  MoveL 3278 to (17.58, -71, -2.56) mm, rotated rx 180 ry 0 rz 90 deg; joints [71.731, -16.979, 81.744, 0, 25.235, 71.731]
  MoveL 3279 to (18.11, -72.42, -2.97) mm, rotated rx -180 ry 0 rz 90 deg; joints [71.692, -16.939, 81.658, 0, 25.28, 71.692]
  MoveL 3280 to (18.93, -73.7, -3.38) mm, rotated rx -180 ry 0 rz 90 deg; joints [71.66, -16.893, 81.554, 0, 25.339, 71.66]
  MoveL 3281 to (20.03, -74.75, -3.78) mm, rotated rx 180 ry 0 rz 90 deg; joints [71.639, -16.843, 81.436, 0, 25.408, 71.639]
  MoveL 3282 to (21.32, -75.54, -4.19) mm, rotated rx 180 ry 0 rz 90 deg; joints [71.627, -16.791, 81.309, 0, 25.482, 71.627]
  MoveL 3283 to (22.76, -76.03, -4.59) mm, rotated rx 180 ry 0 rz 90 deg; joints [71.627, -16.738, 81.179, 0, 25.559, 71.627]
  MoveL 3284 to (24.27, -76.15, -5) mm, rotated rx -180 ry 0 rz 90 deg; joints [71.639, -16.686, 81.052, 0, 25.634, 71.639]
  MoveL 3285 to (45.96, -75.93, -5) mm, rotated rx 180 ry 0 rz 90 deg; joints [71.867, -16.234, 79.464, 0, 26.77, 71.867]
  MoveL 3286 to (52.59, -75.84, -5) mm, rotated rx -180 ry 0 rz 90 deg; joints [71.937, -16.091, 78.973, 0, 27.118, 71.937]
  MoveC 3287 to (55.58, -72.68, -5) mm, rotated rx -180 ry 0 rz 90 deg; joints [72.063, -16.048, 78.827, 0, 27.222, 72.063] to (55.72, -68.34, -5) mm, rotated rx -180 ry 0 rz 90 deg; joints [72.198, -16.076, 78.921, 0, 27.155, 72.198]
  MoveL 3288 to (51.98, -63.97, -5) mm, rotated rx 180 ry 0 rz 90 deg; joints [72.296, -16.187, 79.304, 0, 26.883, 72.296]
  MoveL 3289 to (27.4, -35.54, -5) mm, rotated rx 180 ry 0 rz 90 deg; joints [72.942, -16.885, 81.769, 0, 25.117, 72.942]
  MoveL 3290 to (27.01, -35.1, -5) mm, rotated rx 180 ry 0 rz 90 deg; joints [72.952, -16.896, 81.807, 0, 25.089, 72.952]
  MoveL 3291 to (26.45, -34.59, -5) mm, rotated rx -180 ry 0 rz 90 deg; joints [72.963, -16.91, 81.859, 0, 25.052, 72.963]
  MoveL 3292 to (20.53, -29.85, -5) mm, rotated rx 180 ry 0 rz 90 deg; joints [73.055, -17.057, 82.393, 0, 24.664, 73.055]
  MoveL 3293 to (12.79, -23.65, -5) mm, rotated rx -180 ry 0 rz 90 deg; joints [73.178, -17.244, 83.085, 0, 24.159, 73.178]
  MoveL 3294 to (11.85, -22.94, -5) mm, rotated rx -180 ry 0 rz 90 deg; joints [73.191, -17.267, 83.168, 0, 24.098, 73.191]
  MoveC 3295 to (8.28, -22.05, -5) mm, rotated rx 180 ry 0 rz 90 deg; joints [73.185, -17.34, 83.443, 0, 23.897, 73.185] to (5.13, -23.95, -5) mm, rotated rx 180 ry 0 rz 90 deg; joints [73.094, -17.389, 83.626, 0, 23.763, 73.094]
  MoveC 3296 to (4.8, -24.62, -5) mm, rotated rx -180 ry 0 rz 90 deg; joints [73.069, -17.391, 83.635, 0, 23.756, 73.069] to (4.56, -25.32, -5) mm, rotated rx 180 ry 0 rz 90 deg; joints [73.045, -17.392, 83.637, 0, 23.755, 73.045]
  MoveL 3297 to (-7.48, -70.6, -5) mm, rotated rx 180 ry 0 rz 90 deg; joints [71.481, -17.345, 83.463, 0, 23.882, 71.481]
  MoveC 3298 to (-7, -74.19, -5) mm, rotated rx -180 ry 0 rz 90 deg; joints [71.372, -17.314, 83.344, 0, 23.969, 71.372] to (-4.04, -76.29, -5) mm, rotated rx -180 ry 0 rz 90 deg; joints [71.338, -17.244, 83.084, 0, 24.16, 71.338]
  MoveC 3299 to (-3.21, -76.4, -5) mm, rotated rx 180 ry 0 rz 90 deg; joints [71.343, -17.227, 83.022, 0, 24.205, 71.343] to (-2.37, -76.42, -5) mm, rotated rx 180 ry 0 rz 90 deg; joints [71.351, -17.211, 82.962, 0, 24.249, 71.351]
  MoveL 3300 to (24.27, -76.15, -5) mm, rotated rx -180 ry 0 rz 90 deg; joints [71.639, -16.686, 81.052, 0, 25.634, 71.639]
  MoveL 3301 to (24.2, -68.6, -5) mm, rotated rx -180 ry 0 rz 90 deg; joints [71.873, -16.738, 81.239, 0, 25.5, 71.873]
  MoveL 3302 to (24.2, -68.6, -2) mm, rotated rx 180 ry 0 rz 90 deg; joints [71.873, -16.89, 81.34, 0, 25.55, 71.873]
  Establecer velocidad (1000.0 mm/s)
  MoveL 3303 to (24.2, -68.6, 10) mm, rotated rx -180 ry 0 rz 90 deg; joints [71.873, -17.496, 81.742, 0, 25.754, 71.873]
  Establecer velocidad (66.7 mm/s)
  MoveL 3304 to (66.41, -31.14, 10) mm, rotated rx 180 ry 0 rz 90 deg; joints [73.447, -16.845, 79.487, 0, 27.358, 73.447]
  MoveL 3305 to (66.41, -31.14, -1.75) mm, rotated rx -180 ry 0 rz 90 deg; joints [73.447, -16.257, 79.092, 0, 27.164, 73.447]
  MoveL 3306 to (67.91, -31.32, -2.16) mm, rotated rx -180 ry 0 rz 90 deg; joints [73.456, -16.202, 78.961, 0, 27.241, 73.456]
  MoveL 3307 to (69.42, -31.14, -2.56) mm, rotated rx 180 ry 0 rz 90 deg; joints [73.475, -16.149, 78.838, 0, 27.312, 73.475]
  MoveL 3308 to (70.85, -30.62, -2.97) mm, rotated rx 180 ry 0 rz 90 deg; joints [73.504, -16.101, 78.727, 0, 27.373, 73.504]
  MoveL 3309 to (72.13, -29.81, -3.38) mm, rotated rx -180 ry 0 rz 90 deg; joints [73.541, -16.057, 78.635, 0, 27.422, 73.541]
  MoveL 3310 to (73.2, -28.73, -3.78) mm, rotated rx 180 ry 0 rz 90 deg; joints [73.584, -16.02, 78.564, 0, 27.456, 73.584]
  MoveL 3311 to (74.01, -27.44, -4.19) mm, rotated rx -180 ry 0 rz 90 deg; joints [73.631, -15.99, 78.518, 0, 27.472, 73.631]
  MoveL 3312 to (74.51, -26, -4.59) mm, rotated rx 180 ry 0 rz 90 deg; joints [73.68, -15.968, 78.498, 0, 27.47, 73.68]
  MoveL 3313 to (74.65, -24.49, -5) mm, rotated rx -180 ry 0 rz 90 deg; joints [73.728, -15.954, 78.507, 0, 27.447, 73.728]
  MoveL 3314 to (74.64, -7.37, -5) mm, rotated rx -180 ry 0 rz 90 deg; joints [74.258, -16.064, 78.879, 0, 27.184, 74.258]
  MoveC 3315 to (72.62, -4.69, -5) mm, rotated rx 180 ry 0 rz 90 deg; joints [74.324, -16.125, 79.089, 0, 27.036, 74.324] to (69.65, -3.13, -5) mm, rotated rx -180 ry 0 rz 90 deg; joints [74.346, -16.199, 79.346, 0, 26.854, 74.346]
  MoveC 3316 to (68.13, -3, -5) mm, rotated rx 180 ry 0 rz 90 deg; joints [74.337, -16.233, 79.463, 0, 26.77, 74.337] to (66.64, -3.36, -5) mm, rotated rx -180 ry 0 rz 90 deg; joints [74.313, -16.263, 79.567, 0, 26.696, 74.313]
  MoveL 3317 to (51.96, -23.48, -5) mm, rotated rx -180 ry 0 rz 90 deg; joints [73.552, -16.454, 80.231, 0, 26.223, 73.552]
  MoveC 3318 to (51.14, -26.2, -5) mm, rotated rx -180 ry 0 rz 90 deg; joints [73.46, -16.454, 80.232, 0, 26.222, 73.46] to (52.21, -28.84, -5) mm, rotated rx 180 ry 0 rz 90 deg; joints [73.387, -16.415, 80.094, 0, 26.321, 73.387]
  MoveL 3319 to (67.07, -45.61, -5) mm, rotated rx 180 ry 0 rz 90 deg; joints [73.007, -15.983, 78.603, 0, 27.38, 73.007]
  MoveC 3320 to (69.47, -45.88, -5) mm, rotated rx 180 ry 0 rz 90 deg; joints [73.021, -15.928, 78.416, 0, 27.512, 73.021] to (71.71, -45.01, -5) mm, rotated rx 180 ry 0 rz 90 deg; joints [73.069, -15.883, 78.266, 0, 27.617, 73.069]
  MoveL 3321 to (72.16, -44.7, -5) mm, rotated rx 180 ry 0 rz 90 deg; joints [73.082, -15.875, 78.239, 0, 27.636, 73.082]
  MoveC 3322 to (73.61, -43.33, -5) mm, rotated rx 180 ry 0 rz 90 deg; joints [73.138, -15.852, 78.161, 0, 27.692, 73.138] to (74.63, -41.62, -5) mm, rotated rx 180 ry 0 rz 90 deg; joints [73.2, -15.841, 78.123, 0, 27.718, 73.2]
  MoveL 3323 to (74.65, -41.22, -5) mm, rotated rx -180 ry 0 rz 90 deg; joints [73.212, -15.843, 78.131, 0, 27.713, 73.212]
  MoveL 3324 to (74.65, -24.49, -5) mm, rotated rx -180 ry 0 rz 90 deg; joints [73.728, -15.954, 78.507, 0, 27.447, 73.728]
  MoveL 3325 to (67.09, -24.5, -5) mm, rotated rx 180 ry 0 rz 90 deg; joints [73.659, -16.121, 79.077, 0, 27.044, 73.659]
  MoveL 3326 to (67.09, -24.5, -2) mm, rotated rx -180 ry 0 rz 90 deg; joints [73.659, -16.272, 79.18, 0, 27.092, 73.659]
  Establecer velocidad (1000.0 mm/s)
  MoveL 3327 to (67.09, -24.5, 10) mm, rotated rx -180 ry 0 rz 90 deg; joints [73.659, -16.873, 79.583, 0, 27.29, 73.659]
  Establecer velocidad (66.7 mm/s)
  MoveL 3328 to (37.4, 23.7, 10) mm, rotated rx 180 ry 0 rz 90 deg; joints [74.913, -17.787, 82.786, 0, 25.001, 74.913]
  MoveL 3329 to (37.4, 23.7, -1.75) mm, rotated rx -180 ry 0 rz 90 deg; joints [74.913, -17.192, 82.393, 0, 24.798, 74.913]
  MoveL 3330 to (37.54, 25.21, -2.16) mm, rotated rx -180 ry 0 rz 90 deg; joints [74.963, -17.177, 82.399, 0, 24.778, 74.963]
  MoveL 3331 to (37.32, 26.71, -2.56) mm, rotated rx 180 ry 0 rz 90 deg; joints [75.009, -17.168, 82.431, 0, 24.738, 75.009]
  MoveL 3332 to (36.77, 28.13, -2.97) mm, rotated rx 180 ry 0 rz 90 deg; joints [75.049, -17.166, 82.485, 0, 24.682, 75.049]
  MoveL 3333 to (35.92, 29.39, -3.38) mm, rotated rx -180 ry 0 rz 90 deg; joints [75.082, -17.169, 82.557, 0, 24.612, 75.082]
  MoveL 3334 to (34.81, 30.43, -3.78) mm, rotated rx 180 ry 0 rz 90 deg; joints [75.106, -17.176, 82.645, 0, 24.531, 75.106]
  MoveL 3335 to (33.5, 31.2, -4.19) mm, rotated rx -180 ry 0 rz 90 deg; joints [75.12, -17.185, 82.741, 0, 24.444, 75.12]
  MoveL 3336 to (32.05, 31.66, -4.59) mm, rotated rx 180 ry 0 rz 90 deg; joints [75.122, -17.196, 82.841, 0, 24.354, 75.122]
  MoveL 3337 to (30.54, 31.76, -5) mm, rotated rx 180 ry 0 rz 90 deg; joints [75.113, -17.205, 82.94, 0, 24.266, 75.113]
  MoveL 3338 to (8.05, 31.16, -5) mm, rotated rx 180 ry 0 rz 90 deg; joints [74.898, -17.63, 84.544, 0, 23.085, 74.898]
  MoveL 3339 to (7.58, 31.11, -5) mm, rotated rx 180 ry 0 rz 90 deg; joints [74.893, -17.638, 84.577, 0, 23.061, 74.893]
  MoveC 3340 to (4.29, 29.28, -5) mm, rotated rx 180 ry 0 rz 90 deg; joints [74.804, -17.69, 84.776, 0, 22.914, 74.804] to (3.5, 25.59, -5) mm, rotated rx 180 ry 0 rz 90 deg; joints [74.677, -17.685, 84.76, 0, 22.925, 74.677]
  MoveL 3341 to (3.65, 25.11, -5) mm, rotated rx -180 ry 0 rz 90 deg; joints [74.663, -17.68, 84.741, 0, 22.94, 74.663]
  MoveL 3342 to (9.48, 9, -5) mm, rotated rx 180 ry 0 rz 90 deg; joints [74.194, -17.489, 84.006, 0, 23.483, 74.194]
  MoveL 3343 to (9.79, 8.22, -5) mm, rotated rx 180 ry 0 rz 90 deg; joints [74.171, -17.479, 83.968, 0, 23.511, 74.171]
  MoveC 3344 to (10.34, 7.22, -5) mm, rotated rx -180 ry 0 rz 90 deg; joints [74.144, -17.463, 83.908, 0, 23.555, 74.144] to (11.15, 6.4, -5) mm, rotated rx 180 ry 0 rz 90 deg; joints [74.125, -17.444, 83.834, 0, 23.61, 74.125]
  MoveL 3345 to (27.96, -6.68, -5) mm, rotated rx 180 ry 0 rz 90 deg; joints [73.861, -17.046, 82.353, 0, 24.693, 73.861]
  MoveL 3346 to (28.63, -7.18, -5) mm, rotated rx -180 ry 0 rz 90 deg; joints [73.851, -17.03, 82.294, 0, 24.736, 73.851]
  MoveC 3347 to (31.82, -7.71, -5) mm, rotated rx 180 ry 0 rz 90 deg; joints [73.864, -16.963, 82.05, 0, 24.913, 73.864] to (34.59, -6.03, -5) mm, rotated rx 180 ry 0 rz 90 deg; joints [73.942, -16.917, 81.884, 0, 25.034, 73.942]
  MoveL 3348 to (35.19, -5.21, -5) mm, rotated rx -180 ry 0 rz 90 deg; joints [73.974, -16.91, 81.857, 0, 25.053, 73.974]
  MoveL 3349 to (55.44, 23.03, -5) mm, rotated rx 180 ry 0 rz 90 deg; joints [75.046, -16.655, 80.943, 0, 25.713, 75.046]
  MoveL 3350 to (56.93, 25.11, -5) mm, rotated rx 180 ry 0 rz 90 deg; joints [75.124, -16.636, 80.873, 0, 25.762, 75.124]
  MoveC 3351 to (56.59, 29.37, -5) mm, rotated rx 180 ry 0 rz 90 deg; joints [75.256, -16.666, 80.982, 0, 25.684, 75.256] to (53.5, 32.33, -5) mm, rotated rx -180 ry 0 rz 90 deg; joints [75.325, -16.747, 81.268, 0, 25.478, 75.325]
  MoveL 3352 to (49.75, 32.27, -5) mm, rotated rx -180 ry 0 rz 90 deg; joints [75.291, -16.823, 81.544, 0, 25.279, 75.291]
  MoveL 3353 to (30.54, 31.76, -5) mm, rotated rx 180 ry 0 rz 90 deg; joints [75.113, -17.205, 82.94, 0, 24.266, 75.113]
  MoveL 3354 to (30.74, 24.21, -5) mm, rotated rx -180 ry 0 rz 90 deg; joints [74.872, -17.162, 82.778, 0, 24.383, 74.872]
  MoveL 3355 to (30.74, 24.21, -2) mm, rotated rx -180 ry 0 rz 90 deg; joints [74.872, -17.314, 82.88, 0, 24.434, 74.872]
  Establecer velocidad (1000.0 mm/s)
  MoveL 3356 to (30.74, 24.21, 10) mm, rotated rx -180 ry 0 rz 90 deg; joints [74.872, -17.923, 83.28, 0, 24.643, 74.872]
  Establecer velocidad (66.7 mm/s)
  MoveL 3357 to (25.69, 67.74, 10) mm, rotated rx 180 ry 0 rz 90 deg; joints [76.236, -18.241, 84.456, 0, 23.784, 76.236]
  MoveL 3358 to (25.69, 67.74, -1.75) mm, rotated rx -180 ry 0 rz 90 deg; joints [76.236, -17.642, 84.065, 0, 23.577, 76.236]
  MoveL 3359 to (25.89, 69.24, -2.16) mm, rotated rx -180 ry 0 rz 90 deg; joints [76.287, -17.624, 84.063, 0, 23.561, 76.287]
  MoveL 3360 to (25.73, 70.75, -2.56) mm, rotated rx 180 ry 0 rz 90 deg; joints [76.335, -17.613, 84.088, 0, 23.525, 76.335]
  MoveL 3361 to (25.23, 72.19, -2.97) mm, rotated rx -180 ry 0 rz 90 deg; joints [76.378, -17.609, 84.135, 0, 23.474, 76.378]
  MoveL 3362 to (24.43, 73.48, -3.38) mm, rotated rx 180 ry 0 rz 90 deg; joints [76.413, -17.609, 84.202, 0, 23.407, 76.413]
  MoveL 3363 to (23.36, 74.56, -3.78) mm, rotated rx -180 ry 0 rz 90 deg; joints [76.44, -17.613, 84.284, 0, 23.33, 76.44]
  MoveL 3364 to (22.08, 75.38, -4.19) mm, rotated rx 180 ry 0 rz 90 deg; joints [76.457, -17.62, 84.376, 0, 23.244, 76.457]
  MoveL 3365 to (20.65, 75.89, -4.59) mm, rotated rx -180 ry 0 rz 90 deg; joints [76.463, -17.629, 84.474, 0, 23.155, 76.463]
  MoveL 3366 to (19.14, 76.05, -5) mm, rotated rx -180 ry 0 rz 90 deg; joints [76.456, -17.637, 84.571, 0, 23.065, 76.456]
  MoveL 3367 to (-29.85, 76.54, -5) mm, rotated rx 180 ry 0 rz 90 deg; joints [76.075, -18.492, 88.024, 0, 20.469, 76.075]
  MoveL 3368 to (-31.98, 76.46, -5) mm, rotated rx 180 ry 0 rz 90 deg; joints [76.054, -18.527, 88.169, 0, 20.357, 76.054]
  MoveC 3369 to (-34.9, 72.87, -5) mm, rotated rx 180 ry 0 rz 90 deg; joints [75.909, -18.559, 88.309, 0, 20.251, 75.909] to (-34.36, 68.26, -5) mm, rotated rx 180 ry 0 rz 90 deg; joints [75.758, -18.532, 88.191, 0, 20.341, 75.758]
  MoveL 3370 to (-33.58, 67.76, -5) mm, rotated rx -180 ry 0 rz 90 deg; joints [75.748, -18.517, 88.129, 0, 20.388, 75.748]
  MoveL 3371 to (-11.56, 53.8, -5) mm, rotated rx 180 ry 0 rz 90 deg; joints [75.471, -18.088, 86.352, 0, 21.736, 75.471]
  MoveC 3372 to (-9.41, 52.87, -5) mm, rotated rx 180 ry 0 rz 90 deg; joints [75.459, -18.047, 86.185, 0, 21.862, 75.459] to (-7.08, 52.65, -5) mm, rotated rx 180 ry 0 rz 90 deg; joints [75.471, -18.005, 86.017, 0, 21.988, 75.471]
  MoveL 3373 to (-6.16, 52.71, -5) mm, rotated rx 180 ry 0 rz 90 deg; joints [75.481, -17.989, 85.953, 0, 22.035, 75.481]
  MoveL 3374 to (56.39, 57.32, -5) mm, rotated rx -180 ry 0 rz 90 deg; joints [76.144, -16.818, 81.525, 0, 25.293, 76.144]
  MoveL 3375 to (69.65, 58.51, -5) mm, rotated rx -180 ry 0 rz 90 deg; joints [76.285, -16.547, 80.559, 0, 25.988, 76.285]
  MoveL 3376 to (70.5, 58.62, -5) mm, rotated rx -180 ry 0 rz 90 deg; joints [76.295, -16.53, 80.497, 0, 26.032, 76.295]
  MoveC 3377 to (72.99, 59.89, -5) mm, rotated rx 180 ry 0 rz 90 deg; joints [76.355, -16.483, 80.334, 0, 26.149, 76.355] to (74.04, 62.48, -5) mm, rotated rx 180 ry 0 rz 90 deg; joints [76.445, -16.474, 80.302, 0, 26.172, 76.445]
  MoveL 3378 to (74.05, 63.02, -5) mm, rotated rx -180 ry 0 rz 90 deg; joints [76.462, -16.477, 80.311, 0, 26.166, 76.462]
  MoveL 3379 to (74.05, 70.6, -5) mm, rotated rx 180 ry 0 rz 90 deg; joints [76.703, -16.515, 80.447, 0, 26.068, 76.703]
  MoveL 3380 to (74.03, 71.11, -5) mm, rotated rx 180 ry 0 rz 90 deg; joints [76.719, -16.518, 80.457, 0, 26.061, 76.719]
  MoveC 3381 to (72.87, 73.73, -5) mm, rotated rx -180 ry 0 rz 90 deg; joints [76.793, -16.556, 80.591, 0, 25.965, 76.793] to (70.25, 74.88, -5) mm, rotated rx -180 ry 0 rz 90 deg; joints [76.81, -16.617, 80.808, 0, 25.81, 76.81]
  MoveC 3382 to (46.61, 75.6, -5) mm, rotated rx 180 ry 0 rz 90 deg; joints [76.655, -17.106, 82.572, 0, 24.534, 76.655] to (22.97, 76, -5) mm, rotated rx -180 ry 0 rz 90 deg; joints [76.485, -17.565, 84.296, 0, 23.269, 76.485]
  MoveL 3383 to (19.14, 76.05, -5) mm, rotated rx -180 ry 0 rz 90 deg; joints [76.456, -17.637, 84.571, 0, 23.065, 76.456]
  MoveL 3384 to (19.06, 68.5, -5) mm, rotated rx -180 ry 0 rz 90 deg; joints [76.208, -17.604, 84.445, 0, 23.159, 76.208]
  MoveL 3385 to (19.06, 68.5, -2) mm, rotated rx -180 ry 0 rz 90 deg; joints [76.208, -17.757, 84.547, 0, 23.211, 76.208]
  Establecer velocidad (1000.0 mm/s)
  MoveL 3386 to (19.06, 68.5, 10) mm, rotated rx -180 ry 0 rz 90 deg; joints [76.208, -18.37, 84.946, 0, 23.424, 76.208]
  Establecer velocidad (66.7 mm/s)
  MoveL 3387 to (25.69, 67.49, 10) mm, rotated rx -180 ry 0 rz 90 deg; joints [76.228, -18.239, 84.452, 0, 23.788, 76.228]
  MoveL 3388 to (25.69, 67.49, -2) mm, rotated rx -180 ry 0 rz 90 deg; joints [76.228, -17.628, 84.052, 0, 23.576, 76.228]
  MoveL 3389 to (25.89, 68.99, -2.41) mm, rotated rx 180 ry 0 rz 90 deg; joints [76.279, -17.61, 84.05, 0, 23.56, 76.279]
  MoveL 3390 to (25.73, 70.51, -2.81) mm, rotated rx -180 ry 0 rz 90 deg; joints [76.327, -17.6, 84.075, 0, 23.524, 76.327]
  MoveL 3391 to (25.23, 71.94, -3.22) mm, rotated rx -180 ry 0 rz 90 deg; joints [76.37, -17.595, 84.123, 0, 23.472, 76.37]
  MoveL 3392 to (24.42, 73.23, -3.62) mm, rotated rx -180 ry 0 rz 90 deg; joints [76.405, -17.595, 84.189, 0, 23.406, 76.405]
  MoveL 3393 to (23.36, 74.31, -4.03) mm, rotated rx 180 ry 0 rz 90 deg; joints [76.432, -17.6, 84.271, 0, 23.328, 76.432]
  MoveL 3394 to (22.08, 75.13, -4.44) mm, rotated rx 180 ry 0 rz 90 deg; joints [76.449, -17.606, 84.364, 0, 23.243, 76.449]
  MoveL 3395 to (20.65, 75.64, -4.84) mm, rotated rx 180 ry 0 rz 90 deg; joints [76.454, -17.615, 84.462, 0, 23.153, 76.454]
  MoveL 3396 to (19.14, 75.8, -5.25) mm, rotated rx 180 ry 0 rz 90 deg; joints [76.448, -17.623, 84.559, 0, 23.064, 76.448]
  MoveL 3397 to (-25.11, 76.24, -5.25) mm, rotated rx -180 ry 0 rz 90 deg; joints [76.104, -18.401, 87.683, 0, 20.718, 76.104]
  MoveL 3398 to (-30.8, 76.27, -5.25) mm, rotated rx 180 ry 0 rz 90 deg; joints [76.058, -18.494, 88.076, 0, 20.418, 76.058]
  MoveL 3399 to (-31.4, 76.24, -5.25) mm, rotated rx 180 ry 0 rz 90 deg; joints [76.052, -18.504, 88.117, 0, 20.386, 76.052]
  MoveC 3400 to (-34.26, 72.7, -5.25) mm, rotated rx 180 ry 0 rz 90 deg; joints [75.908, -18.535, 88.253, 0, 20.282, 75.908] to (-33.75, 68.18, -5.25) mm, rotated rx 180 ry 0 rz 90 deg; joints [75.761, -18.509, 88.14, 0, 20.369, 75.761]
  MoveL 3401 to (-33.1, 67.76, -5.25) mm, rotated rx -180 ry 0 rz 90 deg; joints [75.752, -18.497, 88.088, 0, 20.409, 75.752]
  MoveL 3402 to (-11.42, 54, -5.25) mm, rotated rx -180 ry 0 rz 90 deg; joints [75.479, -18.074, 86.337, 0, 21.736, 75.479]
  MoveC 3403 to (-9.3, 53.09, -5.25) mm, rotated rx 180 ry 0 rz 90 deg; joints [75.467, -18.033, 86.172, 0, 21.86, 75.467] to (-7, 52.9, -5.25) mm, rotated rx -180 ry 0 rz 90 deg; joints [75.48, -17.992, 86.007, 0, 21.984, 75.48]
  MoveL 3404 to (45.99, 56.79, -5.25) mm, rotated rx -180 ry 0 rz 90 deg; joints [76.044, -17.014, 82.274, 0, 24.74, 76.044]
  MoveC 3405 to (57.83, 57.75, -5.25) mm, rotated rx 180 ry 0 rz 90 deg; joints [76.169, -16.778, 81.418, 0, 25.36, 76.169] to (69.65, 58.87, -5.25) mm, rotated rx 180 ry 0 rz 90 deg; joints [76.297, -16.536, 80.557, 0, 25.979, 76.297]
  MoveL 3406 to (70.41, 58.98, -5.25) mm, rotated rx 180 ry 0 rz 90 deg; joints [76.306, -16.521, 80.503, 0, 26.018, 76.306]
  MoveC 3407 to (72.7, 60.18, -5.25) mm, rotated rx 180 ry 0 rz 90 deg; joints [76.362, -16.478, 80.352, 0, 26.126, 76.362] to (73.71, 62.58, -5.25) mm, rotated rx -180 ry 0 rz 90 deg; joints [76.445, -16.469, 80.32, 0, 26.149, 76.445]
  MoveL 3408 to (73.73, 63.02, -5.25) mm, rotated rx -180 ry 0 rz 90 deg; joints [76.46, -16.471, 80.326, 0, 26.145, 76.46]
  MoveL 3409 to (73.73, 70.6, -5.25) mm, rotated rx -180 ry 0 rz 90 deg; joints [76.7, -16.509, 80.462, 0, 26.047, 76.7]
  MoveL 3410 to (73.7, 71.06, -5.25) mm, rotated rx 180 ry 0 rz 90 deg; joints [76.715, -16.513, 80.473, 0, 26.039, 76.715]
  MoveC 3411 to (72.55, 73.49, -5.25) mm, rotated rx 180 ry 0 rz 90 deg; joints [76.783, -16.549, 80.602, 0, 25.947, 76.783] to (70.08, 74.55, -5.25) mm, rotated rx 180 ry 0 rz 90 deg; joints [76.799, -16.607, 80.806, 0, 25.801, 76.799]
  MoveC 3412 to (44.76, 75.38, -5.25) mm, rotated rx 180 ry 0 rz 90 deg; joints [76.633, -17.129, 82.695, 0, 24.434, 76.633] to (19.43, 75.79, -5.25) mm, rotated rx -180 ry 0 rz 90 deg; joints [76.45, -17.617, 84.538, 0, 23.08, 76.45]
  MoveL 3413 to (19.14, 75.8, -5.25) mm, rotated rx 180 ry 0 rz 90 deg; joints [76.448, -17.623, 84.559, 0, 23.064, 76.448]
  MoveL 3414 to (19.06, 68.25, -5.25) mm, rotated rx 180 ry 0 rz 90 deg; joints [76.2, -17.59, 84.432, 0, 23.158, 76.2]
  MoveL 3415 to (19.06, 68.25, -2.25) mm, rotated rx -180 ry 0 rz 90 deg; joints [76.2, -17.743, 84.534, 0, 23.21, 76.2]
  Establecer velocidad (1000.0 mm/s)
  MoveL 3416 to (19.06, 68.25, 10) mm, rotated rx -180 ry 0 rz 90 deg; joints [76.2, -18.369, 84.942, 0, 23.427, 76.2]
  Establecer velocidad (66.7 mm/s)
  MoveL 3417 to (37.41, 23.42, 10) mm, rotated rx 180 ry 0 rz 90 deg; joints [74.905, -17.785, 82.78, 0, 25.006, 74.905]
  MoveL 3418 to (37.41, 23.42, -2) mm, rotated rx 180 ry 0 rz 90 deg; joints [74.905, -17.178, 82.379, 0, 24.799, 74.905]
  MoveL 3419 to (37.56, 24.93, -2.41) mm, rotated rx 180 ry 0 rz 90 deg; joints [74.954, -17.162, 82.384, 0, 24.778, 74.954]
  MoveL 3420 to (37.33, 26.44, -2.81) mm, rotated rx 180 ry 0 rz 90 deg; joints [75, -17.154, 82.416, 0, 24.738, 75]
  MoveL 3421 to (36.78, 27.85, -3.22) mm, rotated rx 180 ry 0 rz 90 deg; joints [75.041, -17.152, 82.47, 0, 24.682, 75.041]
  MoveL 3422 to (35.94, 29.11, -3.62) mm, rotated rx -180 ry 0 rz 90 deg; joints [75.074, -17.155, 82.543, 0, 24.612, 75.074]
  MoveL 3423 to (34.83, 30.15, -4.03) mm, rotated rx 180 ry 0 rz 90 deg; joints [75.098, -17.162, 82.63, 0, 24.532, 75.098]
  MoveL 3424 to (33.52, 30.92, -4.44) mm, rotated rx 180 ry 0 rz 90 deg; joints [75.111, -17.171, 82.726, 0, 24.445, 75.111]
  MoveL 3425 to (32.07, 31.39, -4.84) mm, rotated rx 180 ry 0 rz 90 deg; joints [75.114, -17.181, 82.827, 0, 24.354, 75.114]
  MoveL 3426 to (30.56, 31.49, -5.25) mm, rotated rx 180 ry 0 rz 90 deg; joints [75.104, -17.191, 82.925, 0, 24.266, 75.104]
  MoveL 3427 to (8.05, 30.9, -5.25) mm, rotated rx 180 ry 0 rz 90 deg; joints [74.89, -17.616, 84.531, 0, 23.085, 74.89]
  MoveC 3428 to (4.7, 29.22, -5.25) mm, rotated rx 180 ry 0 rz 90 deg; joints [74.806, -17.669, 84.737, 0, 22.932, 74.806] to (3.77, 25.59, -5.25) mm, rotated rx -180 ry 0 rz 90 deg; joints [74.679, -17.668, 84.733, 0, 22.935, 74.679]
  MoveL 3429 to (3.92, 25.11, -5.25) mm, rotated rx 180 ry 0 rz 90 deg; joints [74.665, -17.663, 84.713, 0, 22.95, 74.665]
  MoveL 3430 to (9.96, 8.47, -5.25) mm, rotated rx 180 ry 0 rz 90 deg; joints [74.181, -17.464, 83.952, 0, 23.512, 74.181]
  MoveC 3431 to (10.51, 7.43, -5.25) mm, rotated rx 180 ry 0 rz 90 deg; joints [74.152, -17.448, 83.892, 0, 23.557, 74.152] to (11.34, 6.58, -5.25) mm, rotated rx 180 ry 0 rz 90 deg; joints [74.132, -17.428, 83.816, 0, 23.613, 74.132]
  MoveL 3432 to (27.71, -6.16, -5.25) mm, rotated rx 180 ry 0 rz 90 deg; joints [73.875, -17.041, 82.373, 0, 24.668, 73.875]
  MoveL 3433 to (27.96, -6.35, -5.25) mm, rotated rx -180 ry 0 rz 90 deg; joints [73.871, -17.035, 82.351, 0, 24.684, 73.871]
  MoveL 3434 to (28.9, -7.03, -5.25) mm, rotated rx -180 ry 0 rz 90 deg; joints [73.858, -17.013, 82.268, 0, 24.744, 73.858]
  MoveC 3435 to (32, -7.33, -5.25) mm, rotated rx -180 ry 0 rz 90 deg; joints [73.877, -16.949, 82.037, 0, 24.912, 73.877] to (34.59, -5.61, -5.25) mm, rotated rx 180 ry 0 rz 90 deg; joints [73.956, -16.907, 81.884, 0, 25.023, 73.956]
  MoveL 3436 to (55.44, 23.47, -5.25) mm, rotated rx 180 ry 0 rz 90 deg; joints [75.06, -16.645, 80.943, 0, 25.702, 75.06]
  MoveL 3437 to (56.39, 24.8, -5.25) mm, rotated rx 180 ry 0 rz 90 deg; joints [75.11, -16.633, 80.899, 0, 25.734, 75.11]
  MoveC 3438 to (56.71, 26.56, -5.25) mm, rotated rx 180 ry 0 rz 90 deg; joints [75.168, -16.636, 80.91, 0, 25.726, 75.168] to (56.39, 28.32, -5.25) mm, rotated rx -180 ry 0 rz 90 deg; joints [75.221, -16.652, 80.968, 0, 25.684, 75.221]
  MoveC 3439 to (55.15, 30.57, -5.25) mm, rotated rx -180 ry 0 rz 90 deg; joints [75.282, -16.69, 81.103, 0, 25.587, 75.282] to (53.06, 32.06, -5.25) mm, rotated rx 180 ry 0 rz 90 deg; joints [75.312, -16.742, 81.287, 0, 25.454, 75.312]
  MoveL 3440 to (52.59, 32.06, -5.25) mm, rotated rx 180 ry 0 rz 90 deg; joints [75.308, -16.751, 81.322, 0, 25.429, 75.308]
  MoveL 3441 to (30.56, 31.49, -5.25) mm, rotated rx 180 ry 0 rz 90 deg; joints [75.104, -17.191, 82.925, 0, 24.266, 75.104]
  MoveL 3442 to (30.75, 23.94, -5.25) mm, rotated rx 180 ry 0 rz 90 deg; joints [74.863, -17.147, 82.764, 0, 24.384, 74.863]
  MoveL 3443 to (30.75, 23.94, -2.25) mm, rotated rx 180 ry 0 rz 90 deg; joints [74.863, -17.3, 82.865, 0, 24.435, 74.863]
  Establecer velocidad (1000.0 mm/s)
  MoveL 3444 to (30.75, 23.94, 10) mm, rotated rx 180 ry 0 rz 90 deg; joints [74.863, -17.921, 83.274, 0, 24.647, 74.863]
  Establecer velocidad (66.7 mm/s)
  MoveL 3445 to (66.13, -31.19, 10) mm, rotated rx 180 ry 0 rz 90 deg; joints [73.443, -16.851, 79.507, 0, 27.344, 73.443]
  MoveL 3446 to (66.13, -31.19, -2) mm, rotated rx -180 ry 0 rz 90 deg; joints [73.443, -16.25, 79.103, 0, 27.147, 73.443]
  MoveL 3447 to (67.64, -31.38, -2.41) mm, rotated rx 180 ry 0 rz 90 deg; joints [73.451, -16.195, 78.972, 0, 27.223, 73.451]
  MoveL 3448 to (69.15, -31.2, -2.81) mm, rotated rx -180 ry 0 rz 90 deg; joints [73.471, -16.142, 78.848, 0, 27.294, 73.471]
  MoveL 3449 to (70.58, -30.68, -3.22) mm, rotated rx -180 ry 0 rz 90 deg; joints [73.5, -16.094, 78.738, 0, 27.356, 73.5]
  MoveL 3450 to (71.86, -29.87, -3.62) mm, rotated rx 180 ry 0 rz 90 deg; joints [73.537, -16.05, 78.646, 0, 27.405, 73.537]
  MoveL 3451 to (72.93, -28.79, -4.03) mm, rotated rx 180 ry 0 rz 90 deg; joints [73.58, -16.013, 78.575, 0, 27.438, 73.58]
  MoveL 3452 to (73.73, -27.5, -4.44) mm, rotated rx 180 ry 0 rz 90 deg; joints [73.627, -15.983, 78.529, 0, 27.455, 73.627]
  MoveL 3453 to (74.23, -26.06, -4.84) mm, rotated rx 180 ry 0 rz 90 deg; joints [73.676, -15.961, 78.509, 0, 27.452, 73.676]
  MoveL 3454 to (74.37, -24.55, -5.25) mm, rotated rx 180 ry 0 rz 90 deg; joints [73.723, -15.948, 78.518, 0, 27.43, 73.723]
  MoveL 3455 to (74.37, -8.1, -5.25) mm, rotated rx -180 ry 0 rz 90 deg; joints [74.233, -16.053, 78.876, 0, 27.177, 74.233]
  MoveC 3456 to (72.46, -5.5, -5.25) mm, rotated rx -180 ry 0 rz 90 deg; joints [74.297, -16.111, 79.075, 0, 27.035, 74.297] to (69.65, -3.92, -5.25) mm, rotated rx 180 ry 0 rz 90 deg; joints [74.322, -16.182, 79.321, 0, 26.861, 74.322]
  MoveC 3457 to (68.05, -3.71, -5.25) mm, rotated rx -180 ry 0 rz 90 deg; joints [74.314, -16.218, 79.446, 0, 26.773, 74.314] to (66.47, -4.06, -5.25) mm, rotated rx 180 ry 0 rz 90 deg; joints [74.29, -16.25, 79.557, 0, 26.694, 74.29]
  MoveL 3458 to (66.33, -4.24, -5.25) mm, rotated rx 180 ry 0 rz 90 deg; joints [74.283, -16.252, 79.563, 0, 26.689, 74.283]
  MoveL 3459 to (52.27, -23.5, -5.25) mm, rotated rx -180 ry 0 rz 90 deg; joints [73.555, -16.434, 80.199, 0, 26.236, 73.555]
  MoveC 3460 to (51.46, -26.19, -5.25) mm, rotated rx 180 ry 0 rz 90 deg; joints [73.463, -16.435, 80.199, 0, 26.235, 73.463] to (52.53, -28.79, -5.25) mm, rotated rx 180 ry 0 rz 90 deg; joints [73.392, -16.396, 80.063, 0, 26.333, 73.392]
  MoveL 3461 to (54.31, -30.8, -5.25) mm, rotated rx -180 ry 0 rz 90 deg; joints [73.346, -16.345, 79.886, 0, 26.459, 73.346]
  MoveL 3462 to (66.48, -44.54, -5.25) mm, rotated rx 180 ry 0 rz 90 deg; joints [73.034, -15.99, 78.664, 0, 27.327, 73.034]
  MoveL 3463 to (66.91, -45.01, -5.25) mm, rotated rx -180 ry 0 rz 90 deg; joints [73.024, -15.978, 78.62, 0, 27.357, 73.024]
  MoveC 3464 to (69.16, -45.22, -5.25) mm, rotated rx -180 ry 0 rz 90 deg; joints [73.038, -15.926, 78.445, 0, 27.481, 73.038] to (71.31, -44.49, -5.25) mm, rotated rx 180 ry 0 rz 90 deg; joints [73.081, -15.883, 78.3, 0, 27.583, 73.081]
  MoveC 3465 to (73.1, -42.99, -5.25) mm, rotated rx 180 ry 0 rz 90 deg; joints [73.144, -15.853, 78.199, 0, 27.655, 73.144] to (74.35, -41.01, -5.25) mm, rotated rx 180 ry 0 rz 90 deg; joints [73.216, -15.839, 78.149, 0, 27.689, 73.216]
  MoveL 3466 to (74.37, -40.27, -5.25) mm, rotated rx -180 ry 0 rz 90 deg; joints [73.239, -15.843, 78.165, 0, 27.679, 73.239]
  MoveL 3467 to (74.37, -24.55, -5.25) mm, rotated rx 180 ry 0 rz 90 deg; joints [73.723, -15.948, 78.518, 0, 27.43, 73.723]
  MoveL 3468 to (66.82, -24.55, -5.25) mm, rotated rx -180 ry 0 rz 90 deg; joints [73.655, -16.114, 79.088, 0, 27.026, 73.655]
  MoveL 3469 to (66.82, -24.55, -2.25) mm, rotated rx 180 ry 0 rz 90 deg; joints [73.655, -16.265, 79.19, 0, 27.075, 73.655]
  Establecer velocidad (1000.0 mm/s)
  MoveL 3470 to (66.82, -24.55, 10) mm, rotated rx 180 ry 0 rz 90 deg; joints [73.655, -16.879, 79.602, 0, 27.277, 73.655]
  Establecer velocidad (66.7 mm/s)
  MoveL 3471 to (17.59, -67.73, 10) mm, rotated rx 180 ry 0 rz 90 deg; joints [71.833, -17.636, 82.242, 0, 25.394, 71.833]
  MoveL 3472 to (17.59, -67.73, -2) mm, rotated rx -180 ry 0 rz 90 deg; joints [71.833, -17.029, 81.84, 0, 25.189, 71.833]
  MoveL 3473 to (17.42, -69.24, -2.41) mm, rotated rx -180 ry 0 rz 90 deg; joints [71.784, -17.002, 81.803, 0, 25.199, 71.784]
  MoveL 3474 to (17.61, -70.74, -2.81) mm, rotated rx -180 ry 0 rz 90 deg; joints [71.739, -16.968, 81.739, 0, 25.228, 71.739]
  MoveL 3475 to (18.14, -72.17, -3.22) mm, rotated rx -180 ry 0 rz 90 deg; joints [71.7, -16.927, 81.653, 0, 25.274, 71.7]
  MoveL 3476 to (18.97, -73.44, -3.62) mm, rotated rx 180 ry 0 rz 90 deg; joints [71.669, -16.881, 81.549, 0, 25.332, 71.669]
  MoveL 3477 to (20.06, -74.5, -4.03) mm, rotated rx -180 ry 0 rz 90 deg; joints [71.647, -16.832, 81.431, 0, 25.401, 71.647]
  MoveL 3478 to (21.36, -75.29, -4.44) mm, rotated rx -180 ry 0 rz 90 deg; joints [71.636, -16.78, 81.304, 0, 25.476, 71.636]
  MoveL 3479 to (22.8, -75.78, -4.84) mm, rotated rx 180 ry 0 rz 90 deg; joints [71.635, -16.727, 81.174, 0, 25.553, 71.635]
  MoveL 3480 to (24.31, -75.9, -5.25) mm, rotated rx -180 ry 0 rz 90 deg; joints [71.647, -16.674, 81.047, 0, 25.627, 71.647]
  MoveL 3481 to (42.17, -75.72, -5.25) mm, rotated rx 180 ry 0 rz 90 deg; joints [71.835, -16.304, 79.741, 0, 26.562, 71.835]
  MoveL 3482 to (52.12, -75.59, -5.25) mm, rotated rx 180 ry 0 rz 90 deg; joints [71.94, -16.09, 79.006, 0, 27.085, 71.94]
  MoveC 3483 to (55.04, -72.48, -5.25) mm, rotated rx -180 ry 0 rz 90 deg; joints [72.064, -16.049, 78.863, 0, 27.186, 72.064] to (55.24, -68.23, -5.25) mm, rotated rx 180 ry 0 rz 90 deg; joints [72.197, -16.074, 78.951, 0, 27.124, 72.197]
  MoveL 3484 to (54.92, -67.79, -5.25) mm, rotated rx -180 ry 0 rz 90 deg; joints [72.207, -16.084, 78.985, 0, 27.099, 72.207]
  MoveL 3485 to (53.26, -65.86, -5.25) mm, rotated rx -180 ry 0 rz 90 deg; joints [72.25, -16.134, 79.155, 0, 26.979, 72.25]
  MoveL 3486 to (50.82, -63.02, -5.25) mm, rotated rx 180 ry 0 rz 90 deg; joints [72.314, -16.206, 79.405, 0, 26.802, 72.314]
  MoveL 3487 to (27.08, -35.54, -5.25) mm, rotated rx -180 ry 0 rz 90 deg; joints [72.939, -16.879, 81.783, 0, 25.096, 72.939]
  MoveL 3488 to (27.01, -35.47, -5.25) mm, rotated rx 180 ry 0 rz 90 deg; joints [72.94, -16.881, 81.79, 0, 25.091, 72.94]
  MoveC 3489 to (26.13, -34.67, -5.25) mm, rotated rx 180 ry 0 rz 90 deg; joints [72.957, -16.904, 81.872, 0, 25.032, 72.957] to (25.21, -33.91, -5.25) mm, rotated rx -180 ry 0 rz 90 deg; joints [72.972, -16.927, 81.955, 0, 24.972, 72.972]
  MoveL 3490 to (12.79, -23.97, -5.25) mm, rotated rx 180 ry 0 rz 90 deg; joints [73.168, -17.23, 83.069, 0, 24.16, 73.168]
  MoveL 3491 to (11.85, -23.25, -5.25) mm, rotated rx 180 ry 0 rz 90 deg; joints [73.181, -17.252, 83.153, 0, 24.099, 73.181]
  MoveC 3492 to (8.1, -22.43, -5.25) mm, rotated rx 180 ry 0 rz 90 deg; joints [73.171, -17.329, 83.439, 0, 23.889, 73.171] to (5.03, -24.74, -5.25) mm, rotated rx 180 ry 0 rz 90 deg; joints [73.068, -17.373, 83.608, 0, 23.766, 73.068]
  MoveL 3493 to (4.9, -25.11, -5.25) mm, rotated rx -180 ry 0 rz 90 deg; joints [73.055, -17.374, 83.609, 0, 23.764, 73.055]
  MoveL 3494 to (3.32, -31, -5.25) mm, rotated rx 180 ry 0 rz 90 deg; joints [72.851, -17.369, 83.593, 0, 23.776, 72.851]
  MoveL 3495 to (-7.22, -70.63, -5.25) mm, rotated rx -180 ry 0 rz 90 deg; joints [71.483, -17.328, 83.436, 0, 23.892, 71.483]
  MoveC 3496 to (-6.61, -74.22, -5.25) mm, rotated rx 180 ry 0 rz 90 deg; joints [71.376, -17.293, 83.308, 0, 23.986, 71.376] to (-3.5, -76.1, -5.25) mm, rotated rx -180 ry 0 rz 90 deg; joints [71.35, -17.222, 83.042, 0, 24.18, 71.35]
  MoveL 3497 to (-2.92, -76.16, -5.25) mm, rotated rx -180 ry 0 rz 90 deg; joints [71.354, -17.211, 82.999, 0, 24.211, 71.354]
  MoveL 3498 to (-2.37, -76.17, -5.25) mm, rotated rx 180 ry 0 rz 90 deg; joints [71.359, -17.2, 82.96, 0, 24.24, 71.359]
  MoveL 3499 to (24.31, -75.9, -5.25) mm, rotated rx -180 ry 0 rz 90 deg; joints [71.647, -16.674, 81.047, 0, 25.627, 71.647]
  MoveL 3500 to (24.23, -68.35, -5.25) mm, rotated rx 180 ry 0 rz 90 deg; joints [71.882, -16.727, 81.234, 0, 25.493, 71.882]
  MoveL 3501 to (24.23, -68.35, -2.25) mm, rotated rx 180 ry 0 rz 90 deg; joints [71.882, -16.878, 81.336, 0, 25.543, 71.882]
  Establecer velocidad (1000.0 mm/s)
  MoveL 3502 to (24.23, -68.35, 10) mm, rotated rx -180 ry 0 rz 90 deg; joints [71.882, -17.497, 81.745, 0, 25.751, 71.882]
  Establecer velocidad (66.7 mm/s)
  MoveL 3503 to (-33.52, -52.29, 10) mm, rotated rx -180 ry 0 rz 90 deg; joints [71.79, -18.698, 86.211, 0, 22.487, 71.79]
  MoveL 3504 to (-33.52, -52.29, -2) mm, rotated rx 180 ry 0 rz 90 deg; joints [71.79, -18.082, 85.812, 0, 22.27, 71.79]
  MoveL 3505 to (-32.11, -52.85, -2.41) mm, rotated rx -180 ry 0 rz 90 deg; joints [71.787, -18.033, 85.688, 0, 22.346, 71.787]
  MoveL 3506 to (-30.6, -53.06, -2.81) mm, rotated rx 180 ry 0 rz 90 deg; joints [71.796, -17.985, 85.565, 0, 22.42, 71.796]
  MoveL 3507 to (-29.09, -52.92, -3.22) mm, rotated rx -180 ry 0 rz 90 deg; joints [71.817, -17.938, 85.45, 0, 22.489, 71.817]
  MoveL 3508 to (-27.64, -52.45, -3.62) mm, rotated rx 180 ry 0 rz 90 deg; joints [71.847, -17.894, 85.346, 0, 22.548, 71.847]
  MoveL 3509 to (-26.33, -51.68, -4.03) mm, rotated rx 180 ry 0 rz 90 deg; joints [71.886, -17.855, 85.259, 0, 22.596, 71.886]
  MoveL 3510 to (-25.23, -50.63, -4.44) mm, rotated rx -180 ry 0 rz 90 deg; joints [71.931, -17.82, 85.192, 0, 22.628, 71.931]
  MoveL 3511 to (-24.38, -49.37, -4.84) mm, rotated rx 180 ry 0 rz 90 deg; joints [71.981, -17.792, 85.148, 0, 22.644, 71.981]
  MoveL 3512 to (-23.87, -47.95, -5.25) mm, rotated rx -180 ry 0 rz 90 deg; joints [72.032, -17.77, 85.131, 0, 22.639, 72.032]
  MoveL 3513 to (-17.64, -24.02, -5.25) mm, rotated rx 180 ry 0 rz 90 deg; joints [72.868, -17.794, 85.224, 0, 22.57, 72.868]
  MoveC 3514 to (-17.37, -22.68, -5.25) mm, rotated rx -180 ry 0 rz 90 deg; joints [72.914, -17.796, 85.234, 0, 22.562, 72.914] to (-17.24, -21.33, -5.25) mm, rotated rx -180 ry 0 rz 90 deg; joints [72.959, -17.802, 85.255, 0, 22.547, 72.959]
  MoveC 3515 to (-18.75, -17.75, -5.25) mm, rotated rx -180 ry 0 rz 90 deg; joints [73.06, -17.848, 85.436, 0, 22.412, 73.06] to (-22.44, -16.58, -5.25) mm, rotated rx -180 ry 0 rz 90 deg; joints [73.061, -17.919, 85.718, 0, 22.201, 73.061]
  MoveC 3516 to (-23.55, -16.74, -5.25) mm, rotated rx 180 ry 0 rz 90 deg; joints [73.045, -17.938, 85.792, 0, 22.145, 73.045] to (-24.65, -16.95, -5.25) mm, rotated rx 180 ry 0 rz 90 deg; joints [73.027, -17.956, 85.865, 0, 22.091, 73.027]
  MoveL 3517 to (-72.65, -27.17, -5.25) mm, rotated rx 180 ry 0 rz 90 deg; joints [72.196, -18.691, 88.923, 0, 19.768, 72.196]
  MoveC 3518 to (-75.69, -29.03, -5.25) mm, rotated rx 180 ry 0 rz 90 deg; joints [72.102, -18.728, 89.086, 0, 19.642, 72.102] to (-76.88, -32.39, -5.25) mm, rotated rx 180 ry 0 rz 90 deg; joints [71.977, -18.729, 89.092, 0, 19.637, 71.977]
  MoveL 3519 to (-76.88, -71.03, -5.25) mm, rotated rx 180 ry 0 rz 90 deg; joints [70.701, -18.528, 88.22, 0, 20.308, 70.701]
  MoveC 3520 to (-75.71, -74.29, -5.25) mm, rotated rx 180 ry 0 rz 90 deg; joints [70.608, -18.491, 88.065, 0, 20.426, 70.608] to (-72.74, -76.07, -5.25) mm, rotated rx 180 ry 0 rz 90 deg; joints [70.584, -18.434, 87.824, 0, 20.61, 70.584]
  MoveC 3521 to (-71.85, -76.2, -5.25) mm, rotated rx 180 ry 0 rz 90 deg; joints [70.59, -18.419, 87.761, 0, 20.659, 70.59] to (-70.94, -76.24, -5.25) mm, rotated rx 180 ry 0 rz 90 deg; joints [70.599, -18.405, 87.699, 0, 20.705, 70.599]
  MoveL 3522 to (-42.17, -76.02, -5.25) mm, rotated rx 180 ry 0 rz 90 deg; joints [70.931, -17.926, 85.747, 0, 22.179, 70.931]
  MoveL 3523 to (-35.35, -75.96, -5.25) mm, rotated rx -180 ry 0 rz 90 deg; joints [71.009, -17.808, 85.278, 0, 22.53, 71.009]
  MoveC 3524 to (-32.03, -74.8, -5.25) mm, rotated rx 180 ry 0 rz 90 deg; joints [71.082, -17.756, 85.076, 0, 22.68, 71.082] to (-30.1, -71.87, -5.25) mm, rotated rx 180 ry 0 rz 90 deg; joints [71.197, -17.74, 85.011, 0, 22.728, 71.197]
  MoveL 3525 to (-23.87, -47.95, -5.25) mm, rotated rx -180 ry 0 rz 90 deg; joints [72.032, -17.77, 85.131, 0, 22.639, 72.032]
  MoveL 3526 to (-31.18, -46.04, -5.25) mm, rotated rx 180 ry 0 rz 90 deg; joints [72.017, -17.91, 85.682, 0, 22.228, 72.017]
  MoveL 3527 to (-31.18, -46.04, -2.25) mm, rotated rx -180 ry 0 rz 90 deg; joints [72.017, -18.064, 85.783, 0, 22.281, 72.017]
  Establecer velocidad (1000.0 mm/s)
  MoveL 3528 to (-31.18, -46.04, 10) mm, rotated rx 180 ry 0 rz 90 deg; joints [72.017, -18.693, 86.191, 0, 22.502, 72.017]
  Establecer velocidad (66.7 mm/s)
  MoveL 3529 to (-68.64, 36.24, 10) mm, rotated rx 180 ry 0 rz 90 deg; joints [74.367, -19.716, 90.44, 0, 19.276, 74.367]
  MoveL 3530 to (-68.64, 36.24, -2) mm, rotated rx 180 ry 0 rz 90 deg; joints [74.367, -19.088, 90.04, 0, 19.048, 74.367]
  MoveL 3531 to (-70.14, 36.43, -2.41) mm, rotated rx 180 ry 0 rz 90 deg; joints [74.359, -19.09, 90.131, 0, 18.959, 74.359]
  MoveL 3532 to (-71.65, 36.24, -2.81) mm, rotated rx 180 ry 0 rz 90 deg; joints [74.339, -19.09, 90.215, 0, 18.876, 74.339]
  MoveL 3533 to (-73.08, 35.73, -3.22) mm, rotated rx 180 ry 0 rz 90 deg; joints [74.308, -19.088, 90.287, 0, 18.801, 74.308]
  MoveL 3534 to (-74.37, 34.91, -3.62) mm, rotated rx -180 ry 0 rz 90 deg; joints [74.268, -19.082, 90.344, 0, 18.738, 74.268]
  MoveL 3535 to (-75.44, 33.84, -4.03) mm, rotated rx 180 ry 0 rz 90 deg; joints [74.221, -19.072, 90.381, 0, 18.691, 74.221]
  MoveL 3536 to (-76.24, 32.55, -4.44) mm, rotated rx 180 ry 0 rz 90 deg; joints [74.169, -19.057, 90.397, 0, 18.66, 74.169]
  MoveL 3537 to (-76.74, 31.11, -4.84) mm, rotated rx 180 ry 0 rz 90 deg; joints [74.115, -19.037, 90.389, 0, 18.648, 74.115]
  MoveL 3538 to (-76.88, 29.6, -5.25) mm, rotated rx 180 ry 0 rz 90 deg; joints [74.063, -19.011, 90.356, 0, 18.656, 74.063]
  MoveL 3539 to (-76.88, 1.42, -5.25) mm, rotated rx 180 ry 0 rz 90 deg; joints [73.109, -18.889, 89.802, 0, 19.087, 73.109]
  MoveL 3540 to (-76.87, 0.47, -5.25) mm, rotated rx 180 ry 0 rz 90 deg; joints [73.077, -18.885, 89.783, 0, 19.102, 73.077]
  MoveC 3541 to (-76.47, -1.56, -5.25) mm, rotated rx -180 ry 0 rz 90 deg; joints [73.013, -18.87, 89.714, 0, 19.156, 73.013] to (-75.34, -3.31, -5.25) mm, rotated rx -180 ry 0 rz 90 deg; joints [72.966, -18.845, 89.603, 0, 19.242, 72.966]
  MoveC 3542 to (-73.12, -4.5, -5.25) mm, rotated rx -180 ry 0 rz 90 deg; joints [72.949, -18.806, 89.43, 0, 19.376, 72.949] to (-70.6, -4.6, -5.25) mm, rotated rx -180 ry 0 rz 90 deg; joints [72.971, -18.767, 89.259, 0, 19.508, 72.971]
  MoveL 3543 to (-69.65, -4.41, -5.25) mm, rotated rx 180 ry 0 rz 90 deg; joints [72.987, -18.754, 89.2, 0, 19.554, 72.987]
  MoveL 3544 to (-31.92, 4.26, -5.25) mm, rotated rx -180 ry 0 rz 90 deg; joints [73.651, -18.19, 86.808, 0, 21.381, 73.651]
  MoveL 3545 to (-20.37, 6.93, -5.25) mm, rotated rx -180 ry 0 rz 90 deg; joints [73.848, -18.005, 86.061, 0, 21.944, 73.848]
  MoveL 3546 to (-19.43, 7.24, -5.25) mm, rotated rx -180 ry 0 rz 90 deg; joints [73.868, -17.99, 86.001, 0, 21.989, 73.868]
  MoveC 3547 to (-17.16, 9.04, -5.25) mm, rotated rx 180 ry 0 rz 90 deg; joints [73.948, -17.96, 85.879, 0, 22.08, 73.948] to (-16.33, 11.81, -5.25) mm, rotated rx 180 ry 0 rz 90 deg; joints [74.046, -17.959, 85.877, 0, 22.082, 74.046]
  MoveC 3548 to (-16.45, 13, -5.25) mm, rotated rx 180 ry 0 rz 90 deg; joints [74.084, -17.967, 85.909, 0, 22.058, 74.084] to (-16.76, 14.15, -5.25) mm, rotated rx -180 ry 0 rz 90 deg; joints [74.119, -17.978, 85.953, 0, 22.025, 74.119]
  MoveL 3549 to (-23.46, 32.88, -5.25) mm, rotated rx 180 ry 0 rz 90 deg; joints [74.674, -18.184, 86.785, 0, 21.399, 74.674]
  MoveC 3550 to (-24.37, 34.52, -5.25) mm, rotated rx 180 ry 0 rz 90 deg; joints [74.72, -18.207, 86.879, 0, 21.328, 74.72] to (-25.76, 35.78, -5.25) mm, rotated rx 180 ry 0 rz 90 deg; joints [74.749, -18.236, 86.999, 0, 21.237, 74.749]
  MoveL 3551 to (-67.76, 62.71, -5.25) mm, rotated rx 180 ry 0 rz 90 deg; joints [75.277, -19.011, 90.353, 0, 18.658, 75.277]
  MoveC 3552 to (-69.57, 63.67, -5.25) mm, rotated rx -180 ry 0 rz 90 deg; joints [75.294, -19.041, 90.491, 0, 18.549, 75.294] to (-71.55, 64.23, -5.25) mm, rotated rx -180 ry 0 rz 90 deg; joints [75.295, -19.072, 90.633, 0, 18.438, 75.295]
  MoveC 3553 to (-74.6, 63.6, -5.25) mm, rotated rx -180 ry 0 rz 90 deg; joints [75.246, -19.113, 90.826, 0, 18.287, 75.246] to (-76.51, 61.13, -5.25) mm, rotated rx -180 ry 0 rz 90 deg; joints [75.144, -19.131, 90.91, 0, 18.221, 75.144]
  MoveC 3554 to (-76.79, 59.95, -5.25) mm, rotated rx 180 ry 0 rz 90 deg; joints [75.101, -19.131, 90.907, 0, 18.223, 75.101] to (-76.88, 58.73, -5.25) mm, rotated rx -180 ry 0 rz 90 deg; joints [75.058, -19.127, 90.892, 0, 18.235, 75.058]
  MoveL 3555 to (-76.88, 29.6, -5.25) mm, rotated rx 180 ry 0 rz 90 deg; joints [74.063, -19.011, 90.356, 0, 18.656, 74.063]
  MoveL 3556 to (-69.33, 29.6, -5.25) mm, rotated rx 180 ry 0 rz 90 deg; joints [74.136, -18.9, 89.851, 0, 19.049, 74.136]
  MoveL 3557 to (-69.33, 29.6, -2.25) mm, rotated rx 180 ry 0 rz 90 deg; joints [74.136, -19.057, 89.952, 0, 19.105, 74.136]
  Establecer velocidad (1000.0 mm/s)
  MoveL 3558 to (-69.33, 29.6, 10) mm, rotated rx -180 ry 0 rz 90 deg; joints [74.136, -19.698, 90.361, 0, 19.338, 74.136]
  Establecer velocidad (66.7 mm/s)
  MoveL 3559 to (-68.4, 36.24, 10) mm, rotated rx 180 ry 0 rz 90 deg; joints [74.37, -19.713, 90.424, 0, 19.289, 74.37]
  MoveL 3560 to (-68.4, 36.24, -2.25) mm, rotated rx 180 ry 0 rz 90 deg; joints [74.37, -19.071, 90.015, 0, 19.056, 74.37]
  MoveL 3561 to (-69.9, 36.43, -2.66) mm, rotated rx 180 ry 0 rz 90 deg; joints [74.362, -19.073, 90.106, 0, 18.967, 74.362]
  MoveL 3562 to (-71.41, 36.24, -3.06) mm, rotated rx 180 ry 0 rz 90 deg; joints [74.341, -19.074, 90.19, 0, 18.883, 74.341]
  MoveL 3563 to (-72.84, 35.73, -3.47) mm, rotated rx 180 ry 0 rz 90 deg; joints [74.31, -19.071, 90.262, 0, 18.809, 74.31]
  MoveL 3564 to (-74.12, 34.91, -3.88) mm, rotated rx -180 ry 0 rz 90 deg; joints [74.27, -19.065, 90.319, 0, 18.746, 74.27]
  MoveL 3565 to (-75.19, 33.84, -4.28) mm, rotated rx 180 ry 0 rz 90 deg; joints [74.223, -19.055, 90.356, 0, 18.699, 74.223]
  MoveL 3566 to (-76, 32.55, -4.69) mm, rotated rx 180 ry 0 rz 90 deg; joints [74.171, -19.04, 90.372, 0, 18.668, 74.171]
  MoveL 3567 to (-76.5, 31.11, -5.09) mm, rotated rx 180 ry 0 rz 90 deg; joints [74.118, -19.02, 90.364, 0, 18.656, 74.118]
  MoveL 3568 to (-76.64, 29.6, -5.5) mm, rotated rx 180 ry 0 rz 90 deg; joints [74.065, -18.995, 90.331, 0, 18.663, 74.065]
  MoveL 3569 to (-76.64, 1.42, -5.5) mm, rotated rx 180 ry 0 rz 90 deg; joints [73.112, -18.873, 89.778, 0, 19.095, 73.112]
  MoveL 3570 to (-76.63, 0.47, -5.5) mm, rotated rx -180 ry 0 rz 90 deg; joints [73.08, -18.868, 89.758, 0, 19.11, 73.08]
  MoveC 3571 to (-76.14, -1.73, -5.5) mm, rotated rx 180 ry 0 rz 90 deg; joints [73.011, -18.851, 89.681, 0, 19.17, 73.011] to (-74.74, -3.5, -5.5) mm, rotated rx -180 ry 0 rz 90 deg; joints [72.965, -18.822, 89.551, 0, 19.271, 72.965]
  MoveC 3572 to (-72.75, -4.32, -5.5) mm, rotated rx 180 ry 0 rz 90 deg; joints [72.958, -18.788, 89.401, 0, 19.387, 72.958] to (-70.6, -4.34, -5.5) mm, rotated rx 180 ry 0 rz 90 deg; joints [72.98, -18.756, 89.257, 0, 19.499, 72.98]
  MoveL 3573 to (-69.65, -4.16, -5.5) mm, rotated rx -180 ry 0 rz 90 deg; joints [72.995, -18.742, 89.196, 0, 19.545, 72.995]
  MoveL 3574 to (-37.12, 3.32, -5.5) mm, rotated rx -180 ry 0 rz 90 deg; joints [73.569, -18.259, 87.139, 0, 21.12, 73.569]
  MoveL 3575 to (-20.19, 7.22, -5.5) mm, rotated rx 180 ry 0 rz 90 deg; joints [73.86, -17.991, 86.046, 0, 21.945, 73.86]
  MoveC 3576 to (-17.64, 8.81, -5.5) mm, rotated rx 180 ry 0 rz 90 deg; joints [73.936, -17.954, 85.9, 0, 22.054, 73.936] to (-16.59, 11.62, -5.5) mm, rotated rx 180 ry 0 rz 90 deg; joints [74.038, -17.95, 85.883, 0, 22.067, 74.038]
  MoveC 3577 to (-16.67, 12.82, -5.5) mm, rotated rx 180 ry 0 rz 90 deg; joints [74.076, -17.957, 85.912, 0, 22.045, 74.076] to (-16.97, 14, -5.5) mm, rotated rx -180 ry 0 rz 90 deg; joints [74.112, -17.968, 85.957, 0, 22.012, 74.112]
  MoveL 3578 to (-23.67, 32.78, -5.5) mm, rotated rx 180 ry 0 rz 90 deg; joints [74.669, -18.174, 86.789, 0, 21.385, 74.669]
  MoveC 3579 to (-24.54, 34.34, -5.5) mm, rotated rx -180 ry 0 rz 90 deg; joints [74.713, -18.196, 86.879, 0, 21.317, 74.713] to (-25.87, 35.55, -5.5) mm, rotated rx 180 ry 0 rz 90 deg; joints [74.74, -18.224, 86.994, 0, 21.23, 74.74]
  MoveL 3580 to (-33.64, 40.54, -5.5) mm, rotated rx 180 ry 0 rz 90 deg; joints [74.836, -18.376, 87.625, 0, 20.751, 74.836]
  MoveL 3581 to (-67.94, 62.54, -5.5) mm, rotated rx 180 ry 0 rz 90 deg; joints [75.27, -19, 90.354, 0, 18.646, 75.27]
  MoveC 3582 to (-69.4, 63.32, -5.5) mm, rotated rx 180 ry 0 rz 90 deg; joints [75.284, -19.024, 90.465, 0, 18.559, 75.284] to (-70.96, 63.88, -5.5) mm, rotated rx -180 ry 0 rz 90 deg; joints [75.288, -19.049, 90.58, 0, 18.469, 75.288]
  MoveC 3583 to (-74.14, 63.53, -5.5) mm, rotated rx 180 ry 0 rz 90 deg; joints [75.248, -19.093, 90.786, 0, 18.307, 75.248] to (-76.25, 61.12, -5.5) mm, rotated rx -180 ry 0 rz 90 deg; joints [75.146, -19.114, 90.884, 0, 18.23, 75.146]
  MoveC 3584 to (-76.54, 60.03, -5.5) mm, rotated rx 180 ry 0 rz 90 deg; joints [75.106, -19.114, 90.884, 0, 18.23, 75.106] to (-76.64, 58.9, -5.5) mm, rotated rx -180 ry 0 rz 90 deg; joints [75.066, -19.111, 90.87, 0, 18.241, 75.066]
  MoveL 3585 to (-76.64, 29.6, -5.5) mm, rotated rx 180 ry 0 rz 90 deg; joints [74.065, -18.995, 90.331, 0, 18.663, 74.065]
  MoveL 3586 to (-69.09, 29.6, -5.5) mm, rotated rx 180 ry 0 rz 90 deg; joints [74.138, -18.884, 89.827, 0, 19.057, 74.138]
  MoveL 3587 to (-69.09, 29.6, -2.5) mm, rotated rx 180 ry 0 rz 90 deg; joints [74.138, -19.041, 89.928, 0, 19.113, 74.138]
  Establecer velocidad (1000.0 mm/s)
  MoveL 3588 to (-69.09, 29.6, 10) mm, rotated rx 180 ry 0 rz 90 deg; joints [74.138, -19.695, 90.345, 0, 19.35, 74.138]
  Establecer velocidad (66.7 mm/s)
  MoveL 3589 to (-39.27, -28.73, 10) mm, rotated rx 180 ry 0 rz 90 deg; joints [72.495, -18.931, 87.132, 0, 21.799, 72.495]
  MoveL 3590 to (-39.27, -28.73, -2.25) mm, rotated rx 180 ry 0 rz 90 deg; joints [72.495, -18.299, 86.724, 0, 21.575, 72.495]
  MoveL 3591 to (-39.41, -27.22, -2.66) mm, rotated rx -180 ry 0 rz 90 deg; joints [72.543, -18.288, 86.752, 0, 21.536, 72.543]
  MoveL 3592 to (-39.9, -25.78, -3.06) mm, rotated rx -180 ry 0 rz 90 deg; joints [72.585, -18.283, 86.803, 0, 21.48, 72.585]
  MoveL 3593 to (-40.7, -24.49, -3.47) mm, rotated rx 180 ry 0 rz 90 deg; joints [72.619, -18.283, 86.872, 0, 21.41, 72.619]
  MoveL 3594 to (-41.76, -23.41, -3.88) mm, rotated rx 180 ry 0 rz 90 deg; joints [72.644, -18.285, 86.955, 0, 21.33, 72.644]
  MoveL 3595 to (-43.04, -22.59, -4.28) mm, rotated rx 180 ry 0 rz 90 deg; joints [72.657, -18.29, 87.047, 0, 21.243, 72.657]
  MoveL 3596 to (-44.47, -22.06, -4.69) mm, rotated rx 180 ry 0 rz 90 deg; joints [72.66, -18.295, 87.142, 0, 21.153, 72.66]
  MoveL 3597 to (-45.97, -21.88, -5.09) mm, rotated rx 180 ry 0 rz 90 deg; joints [72.651, -18.3, 87.235, 0, 21.065, 72.651]
  MoveL 3598 to (-47.48, -22.05, -5.5) mm, rotated rx 180 ry 0 rz 90 deg; joints [72.629, -18.303, 87.321, 0, 20.982, 72.629]
  MoveL 3599 to (-72.49, -27.37, -5.5) mm, rotated rx -180 ry 0 rz 90 deg; joints [72.191, -18.674, 88.899, 0, 19.775, 72.191]
  MoveC 3600 to (-74.49, -28.25, -5.5) mm, rotated rx 180 ry 0 rz 90 deg; joints [72.141, -18.7, 89.014, 0, 19.687, 72.141] to (-75.98, -29.85, -5.5) mm, rotated rx 180 ry 0 rz 90 deg; joints [72.072, -18.715, 89.079, 0, 19.636, 72.072]
  MoveC 3601 to (-76.49, -31.23, -5.5) mm, rotated rx 180 ry 0 rz 90 deg; joints [72.02, -18.716, 89.083, 0, 19.633, 72.02] to (-76.64, -32.69, -5.5) mm, rotated rx 180 ry 0 rz 90 deg; joints [71.97, -18.711, 89.061, 0, 19.65, 71.97]
  MoveL 3602 to (-76.64, -70.88, -5.5) mm, rotated rx -180 ry 0 rz 90 deg; joints [70.709, -18.512, 88.199, 0, 20.313, 70.709]
  MoveC 3603 to (-76.3, -72.75, -5.5) mm, rotated rx -180 ry 0 rz 90 deg; joints [70.652, -18.496, 88.132, 0, 20.364, 70.652] to (-75.34, -74.39, -5.5) mm, rotated rx 180 ry 0 rz 90 deg; joints [70.609, -18.472, 88.029, 0, 20.443, 70.609]
  MoveC 3604 to (-73.59, -75.55, -5.5) mm, rotated rx -180 ry 0 rz 90 deg; joints [70.591, -18.438, 87.885, 0, 20.553, 70.591] to (-71.55, -76, -5.5) mm, rotated rx 180 ry 0 rz 90 deg; joints [70.6, -18.403, 87.737, 0, 20.666, 70.6]
  MoveL 3605 to (-70.6, -76.01, -5.5) mm, rotated rx -180 ry 0 rz 90 deg; joints [70.611, -18.387, 87.673, 0, 20.715, 70.611]
  MoveL 3606 to (-42.17, -75.78, -5.5) mm, rotated rx 180 ry 0 rz 90 deg; joints [70.939, -17.915, 85.744, 0, 22.171, 70.939]
  MoveL 3607 to (-35.32, -75.72, -5.5) mm, rotated rx 180 ry 0 rz 90 deg; joints [71.017, -17.796, 85.273, 0, 22.522, 71.017]
  MoveC 3608 to (-32.33, -74.73, -5.5) mm, rotated rx 180 ry 0 rz 90 deg; joints [71.081, -17.749, 85.09, 0, 22.659, 71.081] to (-30.48, -72.19, -5.5) mm, rotated rx -180 ry 0 rz 90 deg; joints [71.183, -17.731, 85.021, 0, 22.71, 71.183]
  MoveC 3609 to (-30.29, -71.59, -5.5) mm, rotated rx -180 ry 0 rz 90 deg; joints [71.204, -17.732, 85.023, 0, 22.709, 71.204] to (-30.12, -71, -5.5) mm, rotated rx 180 ry 0 rz 90 deg; joints [71.225, -17.732, 85.025, 0, 22.707, 71.225]
  MoveL 3610 to (-17.79, -23.67, -5.5) mm, rotated rx -180 ry 0 rz 90 deg; joints [72.877, -17.786, 85.234, 0, 22.552, 72.877]
  MoveC 3611 to (-17.54, -22.31, -5.5) mm, rotated rx 180 ry 0 rz 90 deg; joints [72.924, -17.789, 85.246, 0, 22.543, 72.924] to (-17.52, -20.92, -5.5) mm, rotated rx -180 ry 0 rz 90 deg; joints [72.969, -17.796, 85.274, 0, 22.522, 72.969]
  MoveC 3612 to (-19.1, -17.8, -5.5) mm, rotated rx 180 ry 0 rz 90 deg; joints [73.054, -17.841, 85.451, 0, 22.39, 73.054] to (-22.45, -16.81, -5.5) mm, rotated rx -180 ry 0 rz 90 deg; joints [73.054, -17.905, 85.706, 0, 22.199, 73.054]
  MoveL 3613 to (-23.22, -16.9, -5.5) mm, rotated rx 180 ry 0 rz 90 deg; joints [73.043, -17.918, 85.758, 0, 22.161, 73.043]
  MoveL 3614 to (-47.48, -22.05, -5.5) mm, rotated rx 180 ry 0 rz 90 deg; joints [72.629, -18.303, 87.321, 0, 20.982, 72.629]
  MoveL 3615 to (-45.91, -29.44, -5.5) mm, rotated rx -180 ry 0 rz 90 deg; joints [72.403, -18.239, 87.055, 0, 21.184, 72.403]
  MoveL 3616 to (-45.91, -29.44, -2.5) mm, rotated rx 180 ry 0 rz 90 deg; joints [72.403, -18.394, 87.156, 0, 21.238, 72.403]
  Establecer velocidad (1000.0 mm/s)
  MoveL 3617 to (-45.91, -29.44, 10) mm, rotated rx -180 ry 0 rz 90 deg; joints [72.403, -19.04, 87.572, 0, 21.468, 72.403]
  Establecer velocidad (66.7 mm/s)
  MoveL 3618 to (17.65, -67.49, 10) mm, rotated rx -180 ry 0 rz 90 deg; joints [71.841, -17.636, 82.243, 0, 25.393, 71.841]
  MoveL 3619 to (17.65, -67.49, -2.25) mm, rotated rx 180 ry 0 rz 90 deg; joints [71.841, -17.017, 81.833, 0, 25.184, 71.841]
  MoveL 3620 to (17.48, -68.99, -2.66) mm, rotated rx -180 ry 0 rz 90 deg; joints [71.792, -16.99, 81.796, 0, 25.194, 71.792]
  MoveL 3621 to (17.68, -70.5, -3.06) mm, rotated rx -180 ry 0 rz 90 deg; joints [71.747, -16.955, 81.732, 0, 25.223, 71.747]
  MoveL 3622 to (18.2, -71.93, -3.47) mm, rotated rx -180 ry 0 rz 90 deg; joints [71.708, -16.915, 81.646, 0, 25.269, 71.708]
  MoveL 3623 to (19.03, -73.2, -3.88) mm, rotated rx 180 ry 0 rz 90 deg; joints [71.677, -16.869, 81.542, 0, 25.327, 71.677]
  MoveL 3624 to (20.12, -74.26, -4.28) mm, rotated rx -180 ry 0 rz 90 deg; joints [71.655, -16.819, 81.424, 0, 25.396, 71.655]
  MoveL 3625 to (21.42, -75.05, -4.69) mm, rotated rx 180 ry 0 rz 90 deg; joints [71.644, -16.767, 81.297, 0, 25.471, 71.644]
  MoveL 3626 to (22.86, -75.53, -5.09) mm, rotated rx 180 ry 0 rz 90 deg; joints [71.644, -16.714, 81.167, 0, 25.548, 71.644]
  MoveL 3627 to (24.37, -75.65, -5.5) mm, rotated rx 180 ry 0 rz 90 deg; joints [71.656, -16.662, 81.04, 0, 25.622, 71.656]
  MoveL 3628 to (45.96, -75.42, -5.5) mm, rotated rx 180 ry 0 rz 90 deg; joints [71.883, -16.212, 79.459, 0, 26.753, 71.883]
  MoveL 3629 to (51.65, -75.33, -5.5) mm, rotated rx -180 ry 0 rz 90 deg; joints [71.943, -16.09, 79.039, 0, 27.051, 71.943]
  MoveC 3630 to (54.54, -72.19, -5.5) mm, rotated rx -180 ry 0 rz 90 deg; joints [72.068, -16.049, 78.899, 0, 27.15, 72.068] to (54.68, -67.92, -5.5) mm, rotated rx 180 ry 0 rz 90 deg; joints [72.201, -16.076, 78.991, 0, 27.085, 72.201]
  MoveL 3631 to (51.3, -63.97, -5.5) mm, rotated rx 180 ry 0 rz 90 deg; joints [72.289, -16.177, 79.338, 0, 26.839, 72.289]
  MoveL 3632 to (28.4, -37.43, -5.5) mm, rotated rx -180 ry 0 rz 90 deg; joints [72.892, -16.828, 81.636, 0, 25.192, 72.892]
  MoveL 3633 to (26.75, -35.54, -5.5) mm, rotated rx -180 ry 0 rz 90 deg; joints [72.936, -16.873, 81.799, 0, 25.075, 72.936]
  MoveC 3634 to (26.16, -35, -5.5) mm, rotated rx -180 ry 0 rz 90 deg; joints [72.947, -16.888, 81.853, 0, 25.035, 72.947] to (25.55, -34.49, -5.5) mm, rotated rx -180 ry 0 rz 90 deg; joints [72.957, -16.904, 81.909, 0, 24.995, 72.957]
  MoveL 3635 to (12.65, -24.17, -5.5) mm, rotated rx 180 ry 0 rz 90 deg; joints [73.16, -17.219, 83.067, 0, 24.151, 73.16]
  MoveL 3636 to (11.85, -23.54, -5.5) mm, rotated rx 180 ry 0 rz 90 deg; joints [73.172, -17.238, 83.138, 0, 24.1, 73.172]
  MoveC 3637 to (8.14, -22.79, -5.5) mm, rotated rx 180 ry 0 rz 90 deg; joints [73.16, -17.313, 83.42, 0, 23.893, 73.16] to (5.16, -25.11, -5.5) mm, rotated rx 180 ry 0 rz 90 deg; joints [73.057, -17.356, 83.582, 0, 23.774, 73.057]
  MoveL 3638 to (4.87, -26.06, -5.5) mm, rotated rx -180 ry 0 rz 90 deg; joints [73.024, -17.356, 83.582, 0, 23.774, 73.024]
  MoveL 3639 to (-6.85, -70.23, -5.5) mm, rotated rx 180 ry 0 rz 90 deg; joints [71.499, -17.311, 83.411, 0, 23.9, 71.499]
  MoveC 3640 to (-7, -70.89, -5.5) mm, rotated rx 180 ry 0 rz 90 deg; joints [71.477, -17.309, 83.406, 0, 23.903, 71.477] to (-7.11, -71.55, -5.5) mm, rotated rx 180 ry 0 rz 90 deg; joints [71.455, -17.307, 83.398, 0, 23.909, 71.455]
  MoveC 3641 to (-5.88, -74.58, -5.5) mm, rotated rx 180 ry 0 rz 90 deg; joints [71.372, -17.265, 83.239, 0, 24.026, 71.372] to (-2.9, -75.93, -5.5) mm, rotated rx 180 ry 0 rz 90 deg; joints [71.361, -17.199, 82.995, 0, 24.204, 71.361]
  MoveL 3642 to (-2.37, -75.94, -5.5) mm, rotated rx 180 ry 0 rz 90 deg; joints [71.367, -17.189, 82.957, 0, 24.232, 71.367]
  MoveL 3643 to (24.37, -75.65, -5.5) mm, rotated rx 180 ry 0 rz 90 deg; joints [71.656, -16.662, 81.04, 0, 25.622, 71.656]
  MoveL 3644 to (24.3, -68.11, -5.5) mm, rotated rx -180 ry 0 rz 90 deg; joints [71.89, -16.714, 81.227, 0, 25.488, 71.89]
  MoveL 3645 to (24.3, -68.11, -2.5) mm, rotated rx 180 ry 0 rz 90 deg; joints [71.89, -16.866, 81.328, 0, 25.538, 71.89]
  Establecer velocidad (1000.0 mm/s)
  MoveL 3646 to (24.3, -68.11, 10) mm, rotated rx -180 ry 0 rz 90 deg; joints [71.89, -17.497, 81.747, 0, 25.75, 71.89]
  Establecer velocidad (66.7 mm/s)
  MoveL 3647 to (65.86, -31.19, 10) mm, rotated rx -180 ry 0 rz 90 deg; joints [73.441, -16.857, 79.527, 0, 27.33, 73.441]
  MoveL 3648 to (65.86, -31.19, -2.25) mm, rotated rx -180 ry 0 rz 90 deg; joints [73.441, -16.243, 79.115, 0, 27.128, 73.441]
  MoveL 3649 to (67.37, -31.38, -2.66) mm, rotated rx -180 ry 0 rz 90 deg; joints [73.449, -16.188, 78.984, 0, 27.205, 73.449]
  MoveL 3650 to (68.87, -31.19, -3.06) mm, rotated rx 180 ry 0 rz 90 deg; joints [73.468, -16.136, 78.86, 0, 27.275, 73.468]
  MoveL 3651 to (70.3, -30.68, -3.47) mm, rotated rx -180 ry 0 rz 90 deg; joints [73.497, -16.087, 78.75, 0, 27.337, 73.497]
  MoveL 3652 to (71.59, -29.87, -3.88) mm, rotated rx 180 ry 0 rz 90 deg; joints [73.534, -16.044, 78.658, 0, 27.386, 73.534]
  MoveL 3653 to (72.66, -28.79, -4.28) mm, rotated rx 180 ry 0 rz 90 deg; joints [73.577, -16.007, 78.587, 0, 27.42, 73.577]
  MoveL 3654 to (73.46, -27.5, -4.69) mm, rotated rx 180 ry 0 rz 90 deg; joints [73.624, -15.977, 78.541, 0, 27.436, 73.624]
  MoveL 3655 to (73.96, -26.06, -5.09) mm, rotated rx 180 ry 0 rz 90 deg; joints [73.673, -15.955, 78.521, 0, 27.434, 73.673]
  MoveL 3656 to (74.1, -24.55, -5.5) mm, rotated rx 180 ry 0 rz 90 deg; joints [73.721, -15.941, 78.53, 0, 27.411, 73.721]
  MoveL 3657 to (74.1, -8.83, -5.5) mm, rotated rx -180 ry 0 rz 90 deg; joints [74.208, -16.042, 78.872, 0, 27.169, 74.208]
  MoveC 3658 to (72.3, -6.31, -5.5) mm, rotated rx -180 ry 0 rz 90 deg; joints [74.27, -16.097, 79.062, 0, 27.035, 74.27] to (69.65, -4.71, -5.5) mm, rotated rx 180 ry 0 rz 90 deg; joints [74.297, -16.165, 79.295, 0, 26.869, 74.297]
  MoveC 3659 to (67.97, -4.42, -5.5) mm, rotated rx -180 ry 0 rz 90 deg; joints [74.291, -16.203, 79.428, 0, 26.775, 74.291] to (66.3, -4.75, -5.5) mm, rotated rx 180 ry 0 rz 90 deg; joints [74.266, -16.237, 79.546, 0, 26.691, 74.266]
  MoveL 3660 to (65.96, -5.21, -5.5) mm, rotated rx -180 ry 0 rz 90 deg; joints [74.249, -16.242, 79.562, 0, 26.68, 74.249]
  MoveL 3661 to (52.81, -23.22, -5.5) mm, rotated rx -180 ry 0 rz 90 deg; joints [73.568, -16.412, 80.156, 0, 26.256, 73.568]
  MoveL 3662 to (52.42, -23.81, -5.5) mm, rotated rx 180 ry 0 rz 90 deg; joints [73.546, -16.417, 80.172, 0, 26.245, 73.546]
  MoveC 3663 to (51.79, -26.3, -5.5) mm, rotated rx -180 ry 0 rz 90 deg; joints [73.463, -16.415, 80.164, 0, 26.25, 73.463] to (52.79, -28.66, -5.5) mm, rotated rx -180 ry 0 rz 90 deg; joints [73.398, -16.379, 80.038, 0, 26.34, 73.398]
  MoveL 3664 to (66.33, -43.97, -5.5) mm, rotated rx -180 ry 0 rz 90 deg; joints [73.05, -15.985, 78.679, 0, 27.306, 73.05]
  MoveL 3665 to (66.74, -44.41, -5.5) mm, rotated rx -180 ry 0 rz 90 deg; joints [73.041, -15.973, 78.639, 0, 27.334, 73.041]
  MoveC 3666 to (68.74, -44.66, -5.5) mm, rotated rx -180 ry 0 rz 90 deg; joints [73.052, -15.927, 78.482, 0, 27.445, 73.052] to (70.66, -44.07, -5.5) mm, rotated rx 180 ry 0 rz 90 deg; joints [73.088, -15.888, 78.35, 0, 27.538, 73.088]
  MoveL 3667 to (71.17, -43.77, -5.5) mm, rotated rx -180 ry 0 rz 90 deg; joints [73.102, -15.879, 78.319, 0, 27.56, 73.102]
  MoveC 3668 to (72.93, -42.27, -5.5) mm, rotated rx -180 ry 0 rz 90 deg; joints [73.164, -15.85, 78.22, 0, 27.63, 73.164] to (74.1, -40.27, -5.5) mm, rotated rx -180 ry 0 rz 90 deg; joints [73.236, -15.837, 78.177, 0, 27.66, 73.236]
  MoveL 3669 to (74.1, -24.55, -5.5) mm, rotated rx 180 ry 0 rz 90 deg; joints [73.721, -15.941, 78.53, 0, 27.411, 73.721]
  MoveL 3670 to (66.55, -24.55, -5.5) mm, rotated rx -180 ry 0 rz 90 deg; joints [73.653, -16.108, 79.1, 0, 27.008, 73.653]
  MoveL 3671 to (66.55, -24.55, -2.5) mm, rotated rx 180 ry 0 rz 90 deg; joints [73.653, -16.258, 79.202, 0, 27.056, 73.653]
  Establecer velocidad (1000.0 mm/s)
  MoveL 3672 to (66.55, -24.55, 10) mm, rotated rx 180 ry 0 rz 90 deg; joints [73.653, -16.885, 79.622, 0, 27.262, 73.653]
  Establecer velocidad (66.7 mm/s)
  MoveL 3673 to (37.18, 23.16, 10) mm, rotated rx 180 ry 0 rz 90 deg; joints [74.894, -17.789, 82.792, 0, 24.997, 74.894]
  MoveL 3674 to (37.18, 23.16, -2.25) mm, rotated rx -180 ry 0 rz 90 deg; joints [74.894, -17.168, 82.382, 0, 24.786, 74.894]
  MoveL 3675 to (37.32, 24.67, -2.66) mm, rotated rx -180 ry 0 rz 90 deg; joints [74.944, -17.153, 82.387, 0, 24.765, 74.944]
  MoveL 3676 to (37.1, 26.18, -3.06) mm, rotated rx -180 ry 0 rz 90 deg; joints [74.99, -17.145, 82.42, 0, 24.725, 74.99]
  MoveL 3677 to (36.55, 27.59, -3.47) mm, rotated rx 180 ry 0 rz 90 deg; joints [75.03, -17.142, 82.474, 0, 24.669, 75.03]
  MoveL 3678 to (35.7, 28.85, -3.88) mm, rotated rx 180 ry 0 rz 90 deg; joints [75.064, -17.145, 82.546, 0, 24.599, 75.064]
  MoveL 3679 to (34.59, 29.9, -4.28) mm, rotated rx -180 ry 0 rz 90 deg; joints [75.087, -17.152, 82.633, 0, 24.519, 75.087]
  MoveL 3680 to (33.29, 30.67, -4.69) mm, rotated rx 180 ry 0 rz 90 deg; joints [75.101, -17.162, 82.73, 0, 24.432, 75.101]
  MoveL 3681 to (31.84, 31.13, -5.09) mm, rotated rx -180 ry 0 rz 90 deg; joints [75.103, -17.172, 82.83, 0, 24.342, 75.103]
  MoveL 3682 to (30.33, 31.23, -5.5) mm, rotated rx 180 ry 0 rz 90 deg; joints [75.094, -17.181, 82.928, 0, 24.253, 75.094]
  MoveL 3683 to (8.05, 30.65, -5.5) mm, rotated rx 180 ry 0 rz 90 deg; joints [74.882, -17.602, 84.518, 0, 23.084, 74.882]
  MoveC 3684 to (4.97, 28.97, -5.5) mm, rotated rx 180 ry 0 rz 90 deg; joints [74.8, -17.65, 84.705, 0, 22.945, 74.8] to (4.04, 25.59, -5.5) mm, rotated rx 180 ry 0 rz 90 deg; joints [74.682, -17.65, 84.705, 0, 22.945, 74.682]
  MoveL 3685 to (4.19, 25.11, -5.5) mm, rotated rx 180 ry 0 rz 90 deg; joints [74.668, -17.645, 84.686, 0, 22.959, 74.668]
  MoveL 3686 to (10.17, 8.61, -5.5) mm, rotated rx 180 ry 0 rz 90 deg; joints [74.187, -17.449, 83.932, 0, 23.516, 74.187]
  MoveC 3687 to (10.72, 7.57, -5.5) mm, rotated rx 180 ry 0 rz 90 deg; joints [74.159, -17.433, 83.871, 0, 23.561, 74.159] to (11.55, 6.72, -5.5) mm, rotated rx 180 ry 0 rz 90 deg; joints [74.139, -17.412, 83.795, 0, 23.617, 74.139]
  MoveL 3688 to (27.96, -6.02, -5.5) mm, rotated rx -180 ry 0 rz 90 deg; joints [73.882, -17.024, 82.35, 0, 24.675, 73.882]
  MoveL 3689 to (28.9, -6.71, -5.5) mm, rotated rx -180 ry 0 rz 90 deg; joints [73.869, -17.002, 82.267, 0, 24.735, 73.869]
  MoveC 3690 to (32.01, -6.99, -5.5) mm, rotated rx -180 ry 0 rz 90 deg; joints [73.888, -16.938, 82.035, 0, 24.903, 73.888] to (34.57, -5.21, -5.5) mm, rotated rx -180 ry 0 rz 90 deg; joints [73.968, -16.897, 81.885, 0, 25.012, 73.968]
  MoveL 3691 to (35.26, -4.26, -5.5) mm, rotated rx 180 ry 0 rz 90 deg; joints [74.004, -16.889, 81.855, 0, 25.034, 74.004]
  MoveL 3692 to (55.28, 23.69, -5.5) mm, rotated rx 180 ry 0 rz 90 deg; joints [75.065, -16.637, 80.951, 0, 25.686, 75.065]
  MoveL 3693 to (55.95, 24.64, -5.5) mm, rotated rx -180 ry 0 rz 90 deg; joints [75.101, -16.628, 80.92, 0, 25.709, 75.101]
  MoveC 3694 to (55.62, 28.85, -5.5) mm, rotated rx 180 ry 0 rz 90 deg; joints [75.232, -16.658, 81.027, 0, 25.632, 75.232] to (52.59, 31.79, -5.5) mm, rotated rx 180 ry 0 rz 90 deg; joints [75.3, -16.737, 81.308, 0, 25.429, 75.3]
  MoveL 3695 to (50.7, 31.76, -5.5) mm, rotated rx 180 ry 0 rz 90 deg; joints [75.283, -16.776, 81.448, 0, 25.328, 75.283]
  MoveL 3696 to (30.33, 31.23, -5.5) mm, rotated rx 180 ry 0 rz 90 deg; joints [75.094, -17.181, 82.928, 0, 24.253, 75.094]
  MoveL 3697 to (30.52, 23.68, -5.5) mm, rotated rx -180 ry 0 rz 90 deg; joints [74.853, -17.138, 82.767, 0, 24.371, 74.853]
  MoveL 3698 to (30.52, 23.68, -2.5) mm, rotated rx -180 ry 0 rz 90 deg; joints [74.853, -17.29, 82.868, 0, 24.422, 74.853]
  Establecer velocidad (1000.0 mm/s)
  MoveL 3699 to (30.52, 23.68, 10) mm, rotated rx -180 ry 0 rz 90 deg; joints [74.853, -17.925, 83.286, 0, 24.639, 74.853]
  Establecer velocidad (66.7 mm/s)
  MoveL 3700 to (26.09, 67.25, 10) mm, rotated rx 180 ry 0 rz 90 deg; joints [76.224, -18.231, 84.419, 0, 23.812, 76.224]
  MoveL 3701 to (26.09, 67.25, -2.25) mm, rotated rx -180 ry 0 rz 90 deg; joints [76.224, -17.606, 84.01, 0, 23.596, 76.224]
  MoveL 3702 to (26.29, 68.75, -2.66) mm, rotated rx 180 ry 0 rz 90 deg; joints [76.274, -17.589, 84.009, 0, 23.58, 76.274]
  MoveL 3703 to (26.12, 70.26, -3.06) mm, rotated rx 180 ry 0 rz 90 deg; joints [76.322, -17.578, 84.034, 0, 23.544, 76.322]
  MoveL 3704 to (25.62, 71.69, -3.47) mm, rotated rx -180 ry 0 rz 90 deg; joints [76.365, -17.573, 84.082, 0, 23.492, 76.365]
  MoveL 3705 to (24.82, 72.98, -3.88) mm, rotated rx 180 ry 0 rz 90 deg; joints [76.4, -17.574, 84.148, 0, 23.426, 76.4]
  MoveL 3706 to (23.74, 74.06, -4.28) mm, rotated rx 180 ry 0 rz 90 deg; joints [76.427, -17.578, 84.23, 0, 23.348, 76.427]
  MoveL 3707 to (22.46, 74.88, -4.69) mm, rotated rx 180 ry 0 rz 90 deg; joints [76.444, -17.585, 84.323, 0, 23.262, 76.444]
  MoveL 3708 to (21.03, 75.39, -5.09) mm, rotated rx -180 ry 0 rz 90 deg; joints [76.449, -17.594, 84.421, 0, 23.173, 76.449]
  MoveL 3709 to (19.52, 75.54, -5.5) mm, rotated rx -180 ry 0 rz 90 deg; joints [76.442, -17.602, 84.518, 0, 23.084, 76.442]
  MoveL 3710 to (19.43, 75.54, -5.5) mm, rotated rx -180 ry 0 rz 90 deg; joints [76.442, -17.604, 84.525, 0, 23.078, 76.442]
  MoveL 3711 to (-28.9, 76.05, -5.5) mm, rotated rx 180 ry 0 rz 90 deg; joints [76.066, -18.449, 87.933, 0, 20.516, 76.066]
  MoveL 3712 to (-29.85, 76.05, -5.5) mm, rotated rx -180 ry 0 rz 90 deg; joints [76.058, -18.465, 87.999, 0, 20.466, 76.058]
  MoveL 3713 to (-30.82, 76.02, -5.5) mm, rotated rx 180 ry 0 rz 90 deg; joints [76.049, -18.48, 88.065, 0, 20.415, 76.049]
  MoveC 3714 to (-33.62, 72.52, -5.5) mm, rotated rx -180 ry 0 rz 90 deg; joints [75.908, -18.511, 88.197, 0, 20.314, 75.908] to (-33.13, 68.07, -5.5) mm, rotated rx -180 ry 0 rz 90 deg; joints [75.762, -18.485, 88.086, 0, 20.399, 75.762]
  MoveL 3715 to (-11.21, 54.18, -5.5) mm, rotated rx 180 ry 0 rz 90 deg; joints [75.487, -18.058, 86.318, 0, 21.741, 75.487]
  MoveC 3716 to (-9.2, 53.32, -5.5) mm, rotated rx 180 ry 0 rz 90 deg; joints [75.475, -18.019, 86.161, 0, 21.858, 75.475] to (-7.02, 53.13, -5.5) mm, rotated rx -180 ry 0 rz 90 deg; joints [75.488, -17.98, 86.005, 0, 21.975, 75.488]
  MoveL 3717 to (44.25, 56.92, -5.5) mm, rotated rx -180 ry 0 rz 90 deg; joints [76.035, -17.037, 82.395, 0, 24.642, 76.035]
  MoveC 3718 to (57.14, 57.99, -5.5) mm, rotated rx 180 ry 0 rz 90 deg; joints [76.171, -16.781, 81.465, 0, 25.316, 76.171] to (70.01, 59.27, -5.5) mm, rotated rx 180 ry 0 rz 90 deg; joints [76.312, -16.518, 80.529, 0, 25.989, 76.312]
  MoveC 3719 to (72.44, 60.52, -5.5) mm, rotated rx 180 ry 0 rz 90 deg; joints [76.37, -16.473, 80.37, 0, 26.103, 76.37] to (73.42, 63.07, -5.5) mm, rotated rx 180 ry 0 rz 90 deg; joints [76.459, -16.465, 80.343, 0, 26.123, 76.459]
  MoveL 3720 to (73.42, 70.5, -5.5) mm, rotated rx 180 ry 0 rz 90 deg; joints [76.695, -16.503, 80.476, 0, 26.027, 76.695]
  MoveC 3721 to (72.38, 73.08, -5.5) mm, rotated rx 180 ry 0 rz 90 deg; joints [76.769, -16.538, 80.599, 0, 25.939, 76.769] to (69.85, 74.23, -5.5) mm, rotated rx -180 ry 0 rz 90 deg; joints [76.786, -16.597, 80.809, 0, 25.788, 76.786]
  MoveC 3722 to (44.69, 75.1, -5.5) mm, rotated rx -180 ry 0 rz 90 deg; joints [76.624, -17.116, 82.687, 0, 24.429, 76.624] to (19.52, 75.54, -5.5) mm, rotated rx -180 ry 0 rz 90 deg; joints [76.442, -17.602, 84.518, 0, 23.084, 76.442]
  MoveL 3723 to (19.46, 67.99, -5.5) mm, rotated rx 180 ry 0 rz 90 deg; joints [76.195, -17.569, 84.391, 0, 23.178, 76.195]
  MoveL 3724 to (19.46, 67.99, -2.5) mm, rotated rx 180 ry 0 rz 90 deg; joints [76.195, -17.722, 84.492, 0, 23.23, 76.195]
  Establecer velocidad (1000.0 mm/s)
  MoveL 3725 to (19.46, 67.99, 10) mm, rotated rx -180 ry 0 rz 90 deg; joints [76.195, -18.361, 84.909, 0, 23.452, 76.195]
  Establecer velocidad (66.7 mm/s)
  MoveL 3726 to (26.07, 66.98, 10) mm, rotated rx -180 ry 0 rz 90 deg; joints [76.215, -18.23, 84.416, 0, 23.814, 76.215]
  MoveL 3727 to (26.07, 66.98, -2.5) mm, rotated rx 180 ry 0 rz 90 deg; joints [76.215, -17.593, 83.999, 0, 23.594, 76.215]
  MoveL 3728 to (26.27, 68.49, -2.91) mm, rotated rx -180 ry 0 rz 90 deg; joints [76.266, -17.575, 83.997, 0, 23.578, 76.266]
  MoveL 3729 to (26.11, 70, -3.31) mm, rotated rx 180 ry 0 rz 90 deg; joints [76.313, -17.564, 84.022, 0, 23.542, 76.313]
  MoveL 3730 to (25.61, 71.43, -3.72) mm, rotated rx -180 ry 0 rz 90 deg; joints [76.356, -17.56, 84.069, 0, 23.49, 76.356]
  MoveL 3731 to (24.81, 72.73, -4.12) mm, rotated rx -180 ry 0 rz 90 deg; joints [76.392, -17.56, 84.136, 0, 23.424, 76.392]
  MoveL 3732 to (23.74, 73.81, -4.53) mm, rotated rx -180 ry 0 rz 90 deg; joints [76.419, -17.564, 84.218, 0, 23.346, 76.419]
  MoveL 3733 to (22.46, 74.63, -4.94) mm, rotated rx 180 ry 0 rz 90 deg; joints [76.436, -17.571, 84.311, 0, 23.261, 76.436]
  MoveL 3734 to (21.03, 75.14, -5.34) mm, rotated rx -180 ry 0 rz 90 deg; joints [76.441, -17.58, 84.408, 0, 23.171, 76.441]
  MoveL 3735 to (19.52, 75.3, -5.75) mm, rotated rx -180 ry 0 rz 90 deg; joints [76.434, -17.588, 84.506, 0, 23.082, 76.434]
  MoveL 3736 to (-28.9, 75.82, -5.75) mm, rotated rx -180 ry 0 rz 90 deg; joints [76.058, -18.435, 87.921, 0, 20.514, 76.058]
  MoveL 3737 to (-30.22, 75.8, -5.75) mm, rotated rx -180 ry 0 rz 90 deg; joints [76.047, -18.457, 88.011, 0, 20.445, 76.047]
  MoveC 3738 to (-32.97, 72.34, -5.75) mm, rotated rx -180 ry 0 rz 90 deg; joints [75.907, -18.487, 88.141, 0, 20.346, 75.907] to (-32.49, 67.95, -5.75) mm, rotated rx 180 ry 0 rz 90 deg; joints [75.764, -18.461, 88.032, 0, 20.429, 75.764]
  MoveL 3739 to (-11.1, 54.39, -5.75) mm, rotated rx 180 ry 0 rz 90 deg; joints [75.494, -18.044, 86.306, 0, 21.739, 75.494]
  MoveC 3740 to (-9.16, 53.55, -5.75) mm, rotated rx -180 ry 0 rz 90 deg; joints [75.483, -18.007, 86.154, 0, 21.853, 75.483] to (-7.05, 53.37, -5.75) mm, rotated rx -180 ry 0 rz 90 deg; joints [75.495, -17.969, 86.002, 0, 21.966, 75.495]
  MoveL 3741 to (44.07, 57.15, -5.75) mm, rotated rx 180 ry 0 rz 90 deg; joints [76.041, -17.029, 82.404, 0, 24.625, 76.041]
  MoveL 3742 to (44.82, 57.21, -5.75) mm, rotated rx 180 ry 0 rz 90 deg; joints [76.049, -17.014, 82.35, 0, 24.664, 76.049]
  MoveC 3743 to (57.34, 58.3, -5.75) mm, rotated rx 180 ry 0 rz 90 deg; joints [76.183, -16.765, 81.447, 0, 25.319, 76.183] to (69.85, 59.61, -5.75) mm, rotated rx -180 ry 0 rz 90 deg; joints [76.322, -16.511, 80.539, 0, 25.972, 76.322]
  MoveC 3744 to (72.15, 60.8, -5.75) mm, rotated rx 180 ry 0 rz 90 deg; joints [76.377, -16.468, 80.388, 0, 26.08, 76.377] to (73.09, 63.21, -5.75) mm, rotated rx 180 ry 0 rz 90 deg; joints [76.461, -16.46, 80.361, 0, 26.099, 76.461]
  MoveL 3745 to (73.1, 63.97, -5.75) mm, rotated rx -180 ry 0 rz 90 deg; joints [76.485, -16.464, 80.374, 0, 26.09, 76.485]
  MoveL 3746 to (73.1, 69.65, -5.75) mm, rotated rx 180 ry 0 rz 90 deg; joints [76.665, -16.493, 80.476, 0, 26.017, 76.665]
  MoveL 3747 to (73.09, 70.38, -5.75) mm, rotated rx 180 ry 0 rz 90 deg; joints [76.688, -16.497, 80.49, 0, 26.007, 76.688]
  MoveC 3748 to (72.08, 72.81, -5.75) mm, rotated rx -180 ry 0 rz 90 deg; joints [76.758, -16.53, 80.608, 0, 25.922, 76.758] to (69.68, 73.9, -5.75) mm, rotated rx 180 ry 0 rz 90 deg; joints [76.775, -16.587, 80.807, 0, 25.779, 76.775]
  MoveC 3749 to (45.03, 74.83, -5.75) mm, rotated rx -180 ry 0 rz 90 deg; joints [76.618, -17.095, 82.648, 0, 24.447, 76.618] to (20.37, 75.29, -5.75) mm, rotated rx 180 ry 0 rz 90 deg; joints [76.441, -17.572, 84.444, 0, 23.128, 76.441]
  MoveL 3750 to (19.52, 75.3, -5.75) mm, rotated rx -180 ry 0 rz 90 deg; joints [76.434, -17.588, 84.506, 0, 23.082, 76.434]
  MoveL 3751 to (19.44, 67.75, -5.75) mm, rotated rx 180 ry 0 rz 90 deg; joints [76.187, -17.555, 84.38, 0, 23.176, 76.187]
  MoveL 3752 to (19.44, 67.75, -2.75) mm, rotated rx 180 ry 0 rz 90 deg; joints [76.187, -17.708, 84.481, 0, 23.228, 76.187]
  Establecer velocidad (1000.0 mm/s)
  MoveL 3753 to (19.44, 67.75, 10) mm, rotated rx 180 ry 0 rz 90 deg; joints [76.187, -18.36, 84.906, 0, 23.454, 76.187]
  Establecer velocidad (66.7 mm/s)
  MoveL 3754 to (36.95, 22.91, 10) mm, rotated rx -180 ry 0 rz 90 deg; joints [74.884, -17.792, 82.803, 0, 24.989, 74.884]
  MoveL 3755 to (36.95, 22.91, -2.5) mm, rotated rx -180 ry 0 rz 90 deg; joints [74.884, -17.159, 82.385, 0, 24.774, 74.884]
  MoveL 3756 to (37.1, 24.41, -2.91) mm, rotated rx -180 ry 0 rz 90 deg; joints [74.933, -17.143, 82.39, 0, 24.753, 74.933]
  MoveL 3757 to (36.88, 25.92, -3.31) mm, rotated rx -180 ry 0 rz 90 deg; joints [74.98, -17.135, 82.422, 0, 24.713, 74.98]
  MoveL 3758 to (36.33, 27.34, -3.72) mm, rotated rx -180 ry 0 rz 90 deg; joints [75.02, -17.133, 82.476, 0, 24.657, 75.02]
  MoveL 3759 to (35.48, 28.6, -4.12) mm, rotated rx -180 ry 0 rz 90 deg; joints [75.053, -17.136, 82.549, 0, 24.587, 75.053]
  MoveL 3760 to (34.37, 29.64, -4.53) mm, rotated rx 180 ry 0 rz 90 deg; joints [75.077, -17.143, 82.636, 0, 24.507, 75.077]
  MoveL 3761 to (33.07, 30.41, -4.94) mm, rotated rx 180 ry 0 rz 90 deg; joints [75.091, -17.152, 82.732, 0, 24.419, 75.091]
  MoveL 3762 to (31.62, 30.87, -5.34) mm, rotated rx 180 ry 0 rz 90 deg; joints [75.093, -17.162, 82.833, 0, 24.329, 75.093]
  MoveL 3763 to (30.1, 30.97, -5.75) mm, rotated rx 180 ry 0 rz 90 deg; joints [75.084, -17.171, 82.931, 0, 24.241, 75.084]
  MoveL 3764 to (8.05, 30.41, -5.75) mm, rotated rx -180 ry 0 rz 90 deg; joints [74.874, -17.588, 84.505, 0, 23.083, 74.874]
  MoveC 3765 to (5.08, 28.56, -5.75) mm, rotated rx 180 ry 0 rz 90 deg; joints [74.788, -17.633, 84.68, 0, 22.953, 74.788] to (4.44, 25.11, -5.75) mm, rotated rx -180 ry 0 rz 90 deg; joints [74.67, -17.627, 84.659, 0, 22.969, 74.67]
  MoveL 3766 to (4.78, 24.17, -5.75) mm, rotated rx -180 ry 0 rz 90 deg; joints [74.642, -17.617, 84.617, 0, 23, 74.642]
  MoveL 3767 to (10.38, 8.73, -5.75) mm, rotated rx -180 ry 0 rz 90 deg; joints [74.193, -17.432, 83.911, 0, 23.522, 74.193]
  MoveC 3768 to (10.92, 7.71, -5.75) mm, rotated rx -180 ry 0 rz 90 deg; joints [74.165, -17.417, 83.851, 0, 23.565, 74.165] to (11.72, 6.88, -5.75) mm, rotated rx -180 ry 0 rz 90 deg; joints [74.146, -17.397, 83.777, 0, 23.62, 74.146]
  MoveL 3769 to (27.96, -5.71, -5.75) mm, rotated rx 180 ry 0 rz 90 deg; joints [73.892, -17.014, 82.348, 0, 24.666, 73.892]
  MoveL 3770 to (28.59, -6.16, -5.75) mm, rotated rx -180 ry 0 rz 90 deg; joints [73.883, -16.998, 82.292, 0, 24.706, 73.883]
  MoveC 3771 to (30.61, -6.83, -5.75) mm, rotated rx 180 ry 0 rz 90 deg; joints [73.88, -16.954, 82.131, 0, 24.823, 73.88] to (32.69, -6.38, -5.75) mm, rotated rx 180 ry 0 rz 90 deg; joints [73.914, -16.915, 81.989, 0, 24.926, 73.914]
  MoveL 3772 to (33.15, -6.16, -5.75) mm, rotated rx 180 ry 0 rz 90 deg; joints [73.925, -16.908, 81.961, 0, 24.947, 73.925]
  MoveL 3773 to (33.64, -5.83, -5.75) mm, rotated rx 180 ry 0 rz 90 deg; joints [73.94, -16.9, 81.932, 0, 24.968, 73.94]
  MoveL 3774 to (33.96, -5.53, -5.75) mm, rotated rx 180 ry 0 rz 90 deg; joints [73.952, -16.895, 81.915, 0, 24.98, 73.952]
  MoveL 3775 to (34.26, -5.21, -5.75) mm, rotated rx 180 ry 0 rz 90 deg; joints [73.965, -16.891, 81.899, 0, 24.991, 73.965]
  MoveL 3776 to (34.59, -4.78, -5.75) mm, rotated rx 180 ry 0 rz 90 deg; joints [73.982, -16.887, 81.885, 0, 25.002, 73.982]
  MoveL 3777 to (54.62, 23.22, -5.75) mm, rotated rx 180 ry 0 rz 90 deg; joints [75.045, -16.636, 80.982, 0, 25.654, 75.045]
  MoveL 3778 to (55.44, 24.37, -5.75) mm, rotated rx -180 ry 0 rz 90 deg; joints [75.088, -16.625, 80.944, 0, 25.681, 75.088]
  MoveC 3779 to (55.17, 28.58, -5.75) mm, rotated rx -180 ry 0 rz 90 deg; joints [75.219, -16.654, 81.046, 0, 25.607, 75.219] to (52.15, 31.51, -5.75) mm, rotated rx 180 ry 0 rz 90 deg; joints [75.287, -16.732, 81.327, 0, 25.405, 75.287]
  MoveL 3780 to (49.75, 31.47, -5.75) mm, rotated rx -180 ry 0 rz 90 deg; joints [75.266, -16.781, 81.503, 0, 25.278, 75.266]
  MoveL 3781 to (30.1, 30.97, -5.75) mm, rotated rx 180 ry 0 rz 90 deg; joints [75.084, -17.171, 82.931, 0, 24.241, 75.084]
  MoveL 3782 to (30.3, 23.42, -5.75) mm, rotated rx -180 ry 0 rz 90 deg; joints [74.843, -17.128, 82.77, 0, 24.358, 74.843]
  MoveL 3783 to (30.3, 23.42, -2.75) mm, rotated rx 180 ry 0 rz 90 deg; joints [74.843, -17.28, 82.871, 0, 24.409, 74.843]
  Establecer velocidad (1000.0 mm/s)
  MoveL 3784 to (30.3, 23.42, 10) mm, rotated rx 180 ry 0 rz 90 deg; joints [74.843, -17.928, 83.297, 0, 24.631, 74.843]
  Establecer velocidad (66.7 mm/s)
  MoveL 3785 to (65.59, -31.28, 10) mm, rotated rx 180 ry 0 rz 90 deg; joints [73.435, -16.862, 79.545, 0, 27.317, 73.435]
  MoveL 3786 to (65.59, -31.28, -2.5) mm, rotated rx 180 ry 0 rz 90 deg; joints [73.435, -16.236, 79.125, 0, 27.111, 73.435]
  MoveL 3787 to (67.09, -31.47, -2.91) mm, rotated rx 180 ry 0 rz 90 deg; joints [73.443, -16.181, 78.994, 0, 27.187, 73.443]
  MoveL 3788 to (68.6, -31.28, -3.31) mm, rotated rx -180 ry 0 rz 90 deg; joints [73.463, -16.129, 78.87, 0, 27.258, 73.463]
  MoveL 3789 to (70.03, -30.77, -3.72) mm, rotated rx 180 ry 0 rz 90 deg; joints [73.492, -16.08, 78.76, 0, 27.32, 73.492]
  MoveL 3790 to (71.32, -29.95, -4.12) mm, rotated rx -180 ry 0 rz 90 deg; joints [73.529, -16.037, 78.668, 0, 27.369, 73.529]
  MoveL 3791 to (72.38, -28.87, -4.53) mm, rotated rx -180 ry 0 rz 90 deg; joints [73.572, -16, 78.597, 0, 27.403, 73.572]
  MoveL 3792 to (73.19, -27.58, -4.94) mm, rotated rx 180 ry 0 rz 90 deg; joints [73.619, -15.97, 78.551, 0, 27.419, 73.619]
  MoveL 3793 to (73.69, -26.15, -5.34) mm, rotated rx 180 ry 0 rz 90 deg; joints [73.668, -15.948, 78.531, 0, 27.417, 73.668]
  MoveL 3794 to (73.83, -24.64, -5.75) mm, rotated rx 180 ry 0 rz 90 deg; joints [73.716, -15.934, 78.54, 0, 27.394, 73.716]
  MoveL 3795 to (73.83, -9.55, -5.75) mm, rotated rx -180 ry 0 rz 90 deg; joints [74.183, -16.03, 78.869, 0, 27.162, 74.183]
  MoveC 3796 to (71.67, -6.7, -5.75) mm, rotated rx 180 ry 0 rz 90 deg; joints [74.253, -16.096, 79.093, 0, 27.003, 74.253] to (68.41, -5.21, -5.75) mm, rotated rx -180 ry 0 rz 90 deg; joints [74.271, -16.176, 79.37, 0, 26.806, 74.271]
  MoveC 3797 to (67.26, -5.17, -5.75) mm, rotated rx -180 ry 0 rz 90 deg; joints [74.262, -16.201, 79.457, 0, 26.744, 74.262] to (66.14, -5.45, -5.75) mm, rotated rx 180 ry 0 rz 90 deg; joints [74.243, -16.224, 79.535, 0, 26.688, 74.243]
  MoveL 3798 to (65.86, -5.82, -5.75) mm, rotated rx 180 ry 0 rz 90 deg; joints [74.229, -16.228, 79.548, 0, 26.679, 74.229]
  MoveL 3799 to (52.88, -23.57, -5.75) mm, rotated rx -180 ry 0 rz 90 deg; joints [73.558, -16.396, 80.135, 0, 26.261, 73.558]
  MoveC 3800 to (52.12, -26.19, -5.75) mm, rotated rx 180 ry 0 rz 90 deg; joints [73.469, -16.396, 80.133, 0, 26.262, 73.469] to (53.16, -28.7, -5.75) mm, rotated rx 180 ry 0 rz 90 deg; joints [73.4, -16.358, 80.001, 0, 26.357, 73.4]
  MoveL 3801 to (66.56, -43.8, -5.75) mm, rotated rx 180 ry 0 rz 90 deg; joints [73.058, -15.968, 78.657, 0, 27.311, 73.058]
  MoveC 3802 to (68.85, -43.98, -5.75) mm, rotated rx -180 ry 0 rz 90 deg; joints [73.073, -15.917, 78.481, 0, 27.436, 73.073] to (70.97, -43.12, -5.75) mm, rotated rx 180 ry 0 rz 90 deg; joints [73.12, -15.875, 78.34, 0, 27.535, 73.12]
  MoveL 3803 to (71.22, -42.95, -5.75) mm, rotated rx -180 ry 0 rz 90 deg; joints [73.128, -15.871, 78.325, 0, 27.546, 73.128]
  MoveC 3804 to (72.75, -41.53, -5.75) mm, rotated rx -180 ry 0 rz 90 deg; joints [73.185, -15.846, 78.241, 0, 27.605, 73.185] to (73.82, -39.73, -5.75) mm, rotated rx -180 ry 0 rz 90 deg; joints [73.251, -15.834, 78.202, 0, 27.632, 73.251]
  MoveL 3805 to (73.83, -39.33, -5.75) mm, rotated rx -180 ry 0 rz 90 deg; joints [73.263, -15.837, 78.21, 0, 27.627, 73.263]
  MoveL 3806 to (73.83, -24.64, -5.75) mm, rotated rx 180 ry 0 rz 90 deg; joints [73.716, -15.934, 78.54, 0, 27.394, 73.716]
  MoveL 3807 to (66.28, -24.64, -5.75) mm, rotated rx 180 ry 0 rz 90 deg; joints [73.647, -16.101, 79.11, 0, 26.991, 73.647]
  MoveL 3808 to (66.28, -24.64, -2.75) mm, rotated rx -180 ry 0 rz 90 deg; joints [73.647, -16.251, 79.212, 0, 27.039, 73.647]
  Establecer velocidad (1000.0 mm/s)
  MoveL 3809 to (66.28, -24.64, 10) mm, rotated rx -180 ry 0 rz 90 deg; joints [73.647, -16.89, 79.641, 0, 27.249, 73.647]
  Establecer velocidad (66.7 mm/s)
  MoveL 3810 to (17.55, -67.24, 10) mm, rotated rx 180 ry 0 rz 90 deg; joints [71.848, -17.64, 82.256, 0, 25.384, 71.848]
  MoveL 3811 to (17.55, -67.24, -2.5) mm, rotated rx 180 ry 0 rz 90 deg; joints [71.848, -17.008, 81.838, 0, 25.17, 71.848]
  MoveL 3812 to (17.38, -68.75, -2.91) mm, rotated rx -180 ry 0 rz 90 deg; joints [71.799, -16.981, 81.8, 0, 25.18, 71.799]
  MoveL 3813 to (17.58, -70.26, -3.31) mm, rotated rx 180 ry 0 rz 90 deg; joints [71.754, -16.946, 81.736, 0, 25.21, 71.754]
  MoveL 3814 to (18.11, -71.68, -3.72) mm, rotated rx 180 ry 0 rz 90 deg; joints [71.715, -16.906, 81.65, 0, 25.255, 71.715]
  MoveL 3815 to (18.94, -72.96, -4.12) mm, rotated rx 180 ry 0 rz 90 deg; joints [71.684, -16.86, 81.546, 0, 25.314, 71.684]
  MoveL 3816 to (20.03, -74.01, -4.53) mm, rotated rx -180 ry 0 rz 90 deg; joints [71.662, -16.81, 81.428, 0, 25.383, 71.662]
  MoveL 3817 to (21.33, -74.8, -4.94) mm, rotated rx -180 ry 0 rz 90 deg; joints [71.651, -16.758, 81.301, 0, 25.457, 71.651]
  MoveL 3818 to (22.77, -75.29, -5.34) mm, rotated rx 180 ry 0 rz 90 deg; joints [71.65, -16.705, 81.171, 0, 25.534, 71.65]
  MoveL 3819 to (24.28, -75.41, -5.75) mm, rotated rx 180 ry 0 rz 90 deg; joints [71.662, -16.653, 81.044, 0, 25.609, 71.662]
  MoveL 3820 to (45.96, -75.16, -5.75) mm, rotated rx 180 ry 0 rz 90 deg; joints [71.891, -16.201, 79.457, 0, 26.744, 71.891]
  MoveL 3821 to (51.22, -75.06, -5.75) mm, rotated rx 180 ry 0 rz 90 deg; joints [71.947, -16.089, 79.068, 0, 27.02, 71.947]
  MoveC 3822 to (54.02, -71.94, -5.75) mm, rotated rx 180 ry 0 rz 90 deg; joints [72.071, -16.05, 78.935, 0, 27.115, 72.071] to (54.18, -67.76, -5.75) mm, rotated rx 180 ry 0 rz 90 deg; joints [72.201, -16.076, 79.024, 0, 27.052, 72.201]
  MoveL 3823 to (53.88, -67.37, -5.75) mm, rotated rx 180 ry 0 rz 90 deg; joints [72.21, -16.085, 79.055, 0, 27.029, 72.21]
  MoveL 3824 to (27.01, -36.19, -5.75) mm, rotated rx -180 ry 0 rz 90 deg; joints [72.918, -16.851, 81.757, 0, 25.095, 72.918]
  MoveL 3825 to (26.43, -35.54, -5.75) mm, rotated rx 180 ry 0 rz 90 deg; joints [72.933, -16.867, 81.814, 0, 25.053, 72.933]
  MoveL 3826 to (26.06, -35.2, -5.75) mm, rotated rx -180 ry 0 rz 90 deg; joints [72.94, -16.876, 81.848, 0, 25.029, 72.94]
  MoveL 3827 to (12.27, -24.17, -5.75) mm, rotated rx 180 ry 0 rz 90 deg; joints [73.156, -17.213, 83.085, 0, 24.128, 73.156]
  MoveL 3828 to (11.85, -23.83, -5.75) mm, rotated rx 180 ry 0 rz 90 deg; joints [73.163, -17.223, 83.123, 0, 24.1, 73.163]
  MoveC 3829 to (9.51, -23.02, -5.75) mm, rotated rx 180 ry 0 rz 90 deg; joints [73.166, -17.273, 83.308, 0, 23.964, 73.166] to (7.11, -23.61, -5.75) mm, rotated rx 180 ry 0 rz 90 deg; joints [73.124, -17.315, 83.467, 0, 23.848, 73.124]
  MoveL 3830 to (6.45, -24.06, -5.75) mm, rotated rx 180 ry 0 rz 90 deg; joints [73.103, -17.325, 83.505, 0, 23.82, 73.103]
  MoveC 3831 to (5.66, -24.82, -5.75) mm, rotated rx -180 ry 0 rz 90 deg; joints [73.071, -17.335, 83.544, 0, 23.791, 73.071] to (5.2, -25.81, -5.75) mm, rotated rx -180 ry 0 rz 90 deg; joints [73.035, -17.339, 83.556, 0, 23.783, 73.035]
  MoveL 3832 to (-6.66, -70.38, -5.75) mm, rotated rx 180 ry 0 rz 90 deg; joints [71.497, -17.293, 83.386, 0, 23.908, 71.497]
  MoveC 3833 to (-5.95, -74.02, -5.75) mm, rotated rx 180 ry 0 rz 90 deg; joints [71.389, -17.257, 83.249, 0, 24.008, 71.389] to (-2.66, -75.7, -5.75) mm, rotated rx -180 ry 0 rz 90 deg; joints [71.371, -17.183, 82.975, 0, 24.209, 71.371]
  MoveL 3834 to (-2.37, -75.71, -5.75) mm, rotated rx 180 ry 0 rz 90 deg; joints [71.374, -17.178, 82.954, 0, 24.224, 71.374]
  MoveL 3835 to (24.28, -75.41, -5.75) mm, rotated rx 180 ry 0 rz 90 deg; joints [71.662, -16.653, 81.044, 0, 25.609, 71.662]
  MoveL 3836 to (24.2, -67.86, -5.75) mm, rotated rx 180 ry 0 rz 90 deg; joints [71.897, -16.705, 81.231, 0, 25.474, 71.897]
  MoveL 3837 to (24.2, -67.86, -2.75) mm, rotated rx 180 ry 0 rz 90 deg; joints [71.897, -16.857, 81.333, 0, 25.524, 71.897]
  Establecer velocidad (1000.0 mm/s)
  MoveL 3838 to (24.2, -67.86, 10) mm, rotated rx 180 ry 0 rz 90 deg; joints [71.897, -17.501, 81.76, 0, 25.741, 71.897]
  Establecer velocidad (66.7 mm/s)
  MoveL 3839 to (-33.7, -51.13, 10) mm, rotated rx 180 ry 0 rz 90 deg; joints [71.826, -18.708, 86.25, 0, 22.458, 71.826]
  MoveL 3840 to (-33.7, -51.13, -2.5) mm, rotated rx -180 ry 0 rz 90 deg; joints [71.826, -18.066, 85.834, 0, 22.232, 71.826]
  MoveL 3841 to (-32.29, -51.68, -2.91) mm, rotated rx 180 ry 0 rz 90 deg; joints [71.823, -18.018, 85.71, 0, 22.308, 71.823]
  MoveL 3842 to (-30.78, -51.89, -3.31) mm, rotated rx 180 ry 0 rz 90 deg; joints [71.832, -17.969, 85.587, 0, 22.382, 71.832]
  MoveL 3843 to (-29.27, -51.76, -3.72) mm, rotated rx -180 ry 0 rz 90 deg; joints [71.852, -17.922, 85.472, 0, 22.451, 71.852]
  MoveL 3844 to (-27.82, -51.29, -4.12) mm, rotated rx -180 ry 0 rz 90 deg; joints [71.883, -17.879, 85.368, 0, 22.51, 71.883]
  MoveL 3845 to (-26.51, -50.51, -4.53) mm, rotated rx 180 ry 0 rz 90 deg; joints [71.921, -17.839, 85.281, 0, 22.558, 71.921]
  MoveL 3846 to (-25.41, -49.47, -4.94) mm, rotated rx 180 ry 0 rz 90 deg; joints [71.967, -17.805, 85.214, 0, 22.591, 71.967]
  MoveL 3847 to (-24.56, -48.2, -5.34) mm, rotated rx -180 ry 0 rz 90 deg; joints [72.016, -17.776, 85.17, 0, 22.606, 72.016]
  MoveL 3848 to (-24.05, -46.78, -5.75) mm, rotated rx 180 ry 0 rz 90 deg; joints [72.067, -17.754, 85.153, 0, 22.602, 72.067]
  MoveL 3849 to (-18.1, -23.95, -5.75) mm, rotated rx -180 ry 0 rz 90 deg; joints [72.865, -17.777, 85.241, 0, 22.536, 72.865]
  MoveC 3850 to (-17.87, -22.88, -5.75) mm, rotated rx -180 ry 0 rz 90 deg; joints [72.902, -17.779, 85.248, 0, 22.531, 72.902] to (-17.73, -21.79, -5.75) mm, rotated rx 180 ry 0 rz 90 deg; joints [72.939, -17.782, 85.262, 0, 22.52, 72.939]
  MoveC 3851 to (-19.28, -18.05, -5.75) mm, rotated rx 180 ry 0 rz 90 deg; joints [73.045, -17.83, 85.45, 0, 22.38, 73.045] to (-23.22, -17.13, -5.75) mm, rotated rx -180 ry 0 rz 90 deg; joints [73.036, -17.904, 85.744, 0, 22.16, 73.036]
  MoveL 3852 to (-72.49, -27.61, -5.75) mm, rotated rx 180 ry 0 rz 90 deg; joints [72.183, -18.66, 88.886, 0, 19.774, 72.183]
  MoveC 3853 to (-74.32, -28.42, -5.75) mm, rotated rx -180 ry 0 rz 90 deg; joints [72.137, -18.684, 88.99, 0, 19.693, 72.137] to (-75.71, -29.85, -5.75) mm, rotated rx -180 ry 0 rz 90 deg; joints [72.074, -18.698, 89.052, 0, 19.646, 72.074]
  MoveC 3854 to (-76.24, -31.23, -5.75) mm, rotated rx 180 ry 0 rz 90 deg; joints [72.023, -18.699, 89.058, 0, 19.641, 72.023] to (-76.4, -32.69, -5.75) mm, rotated rx 180 ry 0 rz 90 deg; joints [71.972, -18.694, 89.037, 0, 19.658, 71.972]
  MoveL 3855 to (-76.4, -70.6, -5.75) mm, rotated rx -180 ry 0 rz 90 deg; joints [70.721, -18.496, 88.181, 0, 20.316, 70.721]
  MoveL 3856 to (-76.36, -71.32, -5.75) mm, rotated rx 180 ry 0 rz 90 deg; joints [70.698, -18.492, 88.161, 0, 20.331, 70.698]
  MoveC 3857 to (-76.06, -72.76, -5.75) mm, rotated rx -180 ry 0 rz 90 deg; joints [70.655, -18.479, 88.107, 0, 20.372, 70.655] to (-75.34, -74.04, -5.75) mm, rotated rx -180 ry 0 rz 90 deg; joints [70.621, -18.461, 88.029, 0, 20.432, 70.621]
  MoveC 3858 to (-73.62, -75.29, -5.75) mm, rotated rx 180 ry 0 rz 90 deg; joints [70.6, -18.427, 87.884, 0, 20.542, 70.6] to (-71.55, -75.77, -5.75) mm, rotated rx -180 ry 0 rz 90 deg; joints [70.608, -18.391, 87.734, 0, 20.657, 70.608]
  MoveL 3859 to (-70.6, -75.78, -5.75) mm, rotated rx 180 ry 0 rz 90 deg; joints [70.618, -18.376, 87.67, 0, 20.706, 70.618]
  MoveL 3860 to (-35.36, -75.48, -5.75) mm, rotated rx -180 ry 0 rz 90 deg; joints [71.024, -17.785, 85.273, 0, 22.512, 71.024]
  MoveC 3861 to (-32.32, -74.42, -5.75) mm, rotated rx 180 ry 0 rz 90 deg; joints [71.092, -17.738, 85.088, 0, 22.65, 71.092] to (-30.55, -71.73, -5.75) mm, rotated rx 180 ry 0 rz 90 deg; joints [71.197, -17.723, 85.029, 0, 22.694, 71.197]
  MoveL 3862 to (-24.05, -46.78, -5.75) mm, rotated rx 180 ry 0 rz 90 deg; joints [72.067, -17.754, 85.153, 0, 22.602, 72.067]
  MoveL 3863 to (-31.35, -44.87, -5.75) mm, rotated rx -180 ry 0 rz 90 deg; joints [72.053, -17.894, 85.703, 0, 22.191, 72.053]
  MoveL 3864 to (-31.35, -44.87, -2.75) mm, rotated rx -180 ry 0 rz 90 deg; joints [72.053, -18.048, 85.805, 0, 22.244, 72.053]
  Establecer velocidad (1000.0 mm/s)
  MoveL 3865 to (-31.35, -44.87, 10) mm, rotated rx 180 ry 0 rz 90 deg; joints [72.053, -18.703, 86.229, 0, 22.474, 72.053]
  Establecer velocidad (66.7 mm/s)
  MoveL 3866 to (-68.16, 36.19, 10) mm, rotated rx -180 ry 0 rz 90 deg; joints [74.37, -19.709, 90.407, 0, 19.302, 74.37]
  MoveL 3867 to (-68.16, 36.19, -2.5) mm, rotated rx -180 ry 0 rz 90 deg; joints [74.37, -19.054, 89.99, 0, 19.065, 74.37]
  MoveL 3868 to (-69.66, 36.38, -2.91) mm, rotated rx 180 ry 0 rz 90 deg; joints [74.362, -19.056, 90.081, 0, 18.976, 74.362]
  MoveL 3869 to (-71.17, 36.19, -3.31) mm, rotated rx -180 ry 0 rz 90 deg; joints [74.342, -19.057, 90.165, 0, 18.892, 74.342]
  MoveL 3870 to (-72.6, 35.68, -3.72) mm, rotated rx 180 ry 0 rz 90 deg; joints [74.311, -19.054, 90.237, 0, 18.817, 74.311]
  MoveL 3871 to (-73.88, 34.86, -4.12) mm, rotated rx 180 ry 0 rz 90 deg; joints [74.271, -19.048, 90.294, 0, 18.755, 74.271]
  MoveL 3872 to (-74.95, 33.78, -4.53) mm, rotated rx -180 ry 0 rz 90 deg; joints [74.224, -19.038, 90.331, 0, 18.707, 74.224]
  MoveL 3873 to (-75.76, 32.5, -4.94) mm, rotated rx 180 ry 0 rz 90 deg; joints [74.172, -19.023, 90.347, 0, 18.677, 74.172]
  MoveL 3874 to (-76.26, 31.06, -5.34) mm, rotated rx -180 ry 0 rz 90 deg; joints [74.118, -19.003, 90.339, 0, 18.665, 74.118]
  MoveL 3875 to (-76.4, 29.55, -5.75) mm, rotated rx 180 ry 0 rz 90 deg; joints [74.066, -18.978, 90.306, 0, 18.672, 74.066]
  MoveL 3876 to (-76.4, 1.42, -5.75) mm, rotated rx 180 ry 0 rz 90 deg; joints [73.114, -18.856, 89.753, 0, 19.103, 73.114]
  MoveL 3877 to (-76.39, 0.47, -5.75) mm, rotated rx 180 ry 0 rz 90 deg; joints [73.082, -18.851, 89.733, 0, 19.118, 73.082]
  MoveC 3878 to (-75.92, -1.63, -5.75) mm, rotated rx -180 ry 0 rz 90 deg; joints [73.016, -18.835, 89.659, 0, 19.176, 73.016] to (-74.57, -3.32, -5.75) mm, rotated rx 180 ry 0 rz 90 deg; joints [72.973, -18.807, 89.535, 0, 19.272, 72.973]
  MoveC 3879 to (-72.66, -4.1, -5.75) mm, rotated rx 180 ry 0 rz 90 deg; joints [72.966, -18.775, 89.391, 0, 19.384, 72.966] to (-70.6, -4.11, -5.75) mm, rotated rx 180 ry 0 rz 90 deg; joints [72.987, -18.743, 89.252, 0, 19.491, 72.987]
  MoveL 3880 to (-69.65, -3.94, -5.75) mm, rotated rx 180 ry 0 rz 90 deg; joints [73.003, -18.73, 89.193, 0, 19.537, 73.003]
  MoveL 3881 to (-59.23, -1.53, -5.75) mm, rotated rx 180 ry 0 rz 90 deg; joints [73.189, -18.58, 88.54, 0, 20.04, 73.189]
  MoveL 3882 to (-20.37, 7.41, -5.75) mm, rotated rx 180 ry 0 rz 90 deg; joints [73.864, -17.982, 86.054, 0, 21.928, 73.864]
  MoveC 3883 to (-17.52, 9.38, -5.75) mm, rotated rx -180 ry 0 rz 90 deg; joints [73.956, -17.942, 85.895, 0, 22.047, 73.956] to (-16.89, 12.79, -5.75) mm, rotated rx -180 ry 0 rz 90 deg; joints [74.073, -17.948, 85.919, 0, 22.029, 74.073]
  MoveL 3884 to (-17.11, 13.74, -5.75) mm, rotated rx 180 ry 0 rz 90 deg; joints [74.102, -17.957, 85.953, 0, 22.003, 74.102]
  MoveL 3885 to (-23.89, 32.69, -5.75) mm, rotated rx 180 ry 0 rz 90 deg; joints [74.664, -18.164, 86.794, 0, 21.37, 74.664]
  MoveC 3886 to (-24.59, 34.01, -5.75) mm, rotated rx 180 ry 0 rz 90 deg; joints [74.701, -18.182, 86.868, 0, 21.315, 74.701] to (-25.6, 35.11, -5.75) mm, rotated rx 180 ry 0 rz 90 deg; joints [74.728, -18.205, 86.959, 0, 21.246, 74.728]
  MoveL 3887 to (-68.07, 62.35, -5.75) mm, rotated rx -180 ry 0 rz 90 deg; joints [75.262, -18.988, 90.351, 0, 18.637, 75.262]
  MoveC 3888 to (-69.43, 63.09, -5.75) mm, rotated rx -180 ry 0 rz 90 deg; joints [75.275, -19.01, 90.454, 0, 18.556, 75.275] to (-70.87, 63.62, -5.75) mm, rotated rx -180 ry 0 rz 90 deg; joints [75.28, -19.033, 90.561, 0, 18.473, 75.28]
  MoveC 3889 to (-74.18, 63.21, -5.75) mm, rotated rx 180 ry 0 rz 90 deg; joints [75.237, -19.079, 90.774, 0, 18.305, 75.237] to (-76.17, 60.54, -5.75) mm, rotated rx -180 ry 0 rz 90 deg; joints [75.127, -19.098, 90.86, 0, 18.238, 75.127]
  MoveC 3890 to (-76.34, 59.59, -5.75) mm, rotated rx 180 ry 0 rz 90 deg; joints [75.093, -19.096, 90.854, 0, 18.242, 75.093] to (-76.4, 58.63, -5.75) mm, rotated rx -180 ry 0 rz 90 deg; joints [75.059, -19.094, 90.841, 0, 18.253, 75.059]
  MoveL 3891 to (-76.4, 29.55, -5.75) mm, rotated rx 180 ry 0 rz 90 deg; joints [74.066, -18.978, 90.306, 0, 18.672, 74.066]
  MoveL 3892 to (-68.85, 29.55, -5.75) mm, rotated rx 180 ry 0 rz 90 deg; joints [74.139, -18.867, 89.801, 0, 19.066, 74.139]
  MoveL 3893 to (-68.85, 29.55, -2.75) mm, rotated rx 180 ry 0 rz 90 deg; joints [74.139, -19.024, 89.902, 0, 19.121, 74.139]
  Establecer velocidad (1000.0 mm/s)
  MoveL 3894 to (-68.85, 29.55, 10) mm, rotated rx -180 ry 0 rz 90 deg; joints [74.139, -19.691, 90.327, 0, 19.364, 74.139]
  Establecer velocidad (66.7 mm/s)
  MoveL 3895 to (-67.93, 36.19, 10) mm, rotated rx 180 ry 0 rz 90 deg; joints [74.372, -19.706, 90.392, 0, 19.314, 74.372]
  MoveL 3896 to (-67.93, 36.19, -2.75) mm, rotated rx 180 ry 0 rz 90 deg; joints [74.372, -19.038, 89.967, 0, 19.071, 74.372]
  MoveL 3897 to (-69.44, 36.38, -3.16) mm, rotated rx 180 ry 0 rz 90 deg; joints [74.364, -19.04, 90.057, 0, 18.982, 74.364]
  MoveL 3898 to (-70.95, 36.19, -3.56) mm, rotated rx 180 ry 0 rz 90 deg; joints [74.344, -19.04, 90.141, 0, 18.899, 74.344]
  MoveL 3899 to (-72.38, 35.68, -3.97) mm, rotated rx 180 ry 0 rz 90 deg; joints [74.313, -19.038, 90.214, 0, 18.824, 74.313]
  MoveL 3900 to (-73.66, 34.86, -4.37) mm, rotated rx 180 ry 0 rz 90 deg; joints [74.273, -19.032, 90.27, 0, 18.762, 74.273]
  MoveL 3901 to (-74.73, 33.78, -4.78) mm, rotated rx 180 ry 0 rz 90 deg; joints [74.226, -19.022, 90.308, 0, 18.714, 74.226]
  MoveL 3902 to (-75.53, 32.5, -5.19) mm, rotated rx 180 ry 0 rz 90 deg; joints [74.174, -19.007, 90.323, 0, 18.684, 74.174]
  MoveL 3903 to (-76.03, 31.06, -5.59) mm, rotated rx 180 ry 0 rz 90 deg; joints [74.121, -18.987, 90.316, 0, 18.671, 74.121]
  MoveL 3904 to (-76.17, 29.55, -6) mm, rotated rx -180 ry 0 rz 90 deg; joints [74.068, -18.962, 90.283, 0, 18.679, 74.068]
  MoveL 3905 to (-76.17, 1.42, -6) mm, rotated rx 180 ry 0 rz 90 deg; joints [73.116, -18.84, 89.73, 0, 19.11, 73.116]
  MoveL 3906 to (-76.16, 0.47, -6) mm, rotated rx 180 ry 0 rz 90 deg; joints [73.084, -18.835, 89.71, 0, 19.125, 73.084]
  MoveC 3907 to (-74.83, -2.77, -6) mm, rotated rx 180 ry 0 rz 90 deg; joints [72.989, -18.801, 89.555, 0, 19.245, 72.989] to (-71.54, -3.97, -6) mm, rotated rx -180 ry 0 rz 90 deg; joints [72.982, -18.745, 89.31, 0, 19.435, 72.982]
  MoveC 3908 to (-70.61, -3.87, -6) mm, rotated rx 180 ry 0 rz 90 deg; joints [72.995, -18.732, 89.25, 0, 19.482, 72.995] to (-69.7, -3.7, -6) mm, rotated rx -180 ry 0 rz 90 deg; joints [73.01, -18.719, 89.192, 0, 19.527, 73.01]
  MoveL 3909 to (-20.37, 7.64, -6) mm, rotated rx -180 ry 0 rz 90 deg; joints [73.872, -17.97, 86.05, 0, 21.92, 73.872]
  MoveC 3910 to (-17.69, 9.55, -6) mm, rotated rx -180 ry 0 rz 90 deg; joints [73.96, -17.933, 85.901, 0, 22.032, 73.96] to (-17.11, 12.8, -6) mm, rotated rx 180 ry 0 rz 90 deg; joints [74.071, -17.939, 85.926, 0, 22.013, 74.071]
  MoveC 3911 to (-17.29, 13.51, -6) mm, rotated rx 180 ry 0 rz 90 deg; joints [74.093, -17.946, 85.953, 0, 21.993, 74.093] to (-17.51, 14.2, -6) mm, rotated rx 180 ry 0 rz 90 deg; joints [74.114, -17.953, 85.982, 0, 21.971, 74.114]
  MoveL 3912 to (-18.48, 16.87, -6) mm, rotated rx -180 ry 0 rz 90 deg; joints [74.192, -17.983, 86.102, 0, 21.881, 74.192]
  MoveL 3913 to (-23.45, 30.8, -6) mm, rotated rx 180 ry 0 rz 90 deg; joints [74.605, -18.135, 86.719, 0, 21.416, 74.605]
  MoveL 3914 to (-24.15, 32.71, -6) mm, rotated rx 180 ry 0 rz 90 deg; joints [74.662, -18.156, 86.804, 0, 21.352, 74.662]
  MoveC 3915 to (-24.92, 34.1, -6) mm, rotated rx 180 ry 0 rz 90 deg; joints [74.701, -18.175, 86.884, 0, 21.292, 74.701] to (-26.1, 35.16, -6) mm, rotated rx -180 ry 0 rz 90 deg; joints [74.726, -18.2, 86.986, 0, 21.215, 74.726]
  MoveL 3916 to (-68.18, 62.16, -6) mm, rotated rx -180 ry 0 rz 90 deg; joints [75.255, -18.975, 90.346, 0, 18.629, 75.255]
  MoveC 3917 to (-69.36, 62.81, -6) mm, rotated rx -180 ry 0 rz 90 deg; joints [75.266, -18.995, 90.436, 0, 18.559, 75.266] to (-70.6, 63.31, -6) mm, rotated rx -180 ry 0 rz 90 deg; joints [75.272, -19.015, 90.529, 0, 18.486, 75.272]
  MoveC 3918 to (-73.77, 63.09, -6) mm, rotated rx -180 ry 0 rz 90 deg; joints [75.236, -19.06, 90.736, 0, 18.324, 75.236] to (-75.9, 60.74, -6) mm, rotated rx -180 ry 0 rz 90 deg; joints [75.136, -19.081, 90.837, 0, 18.245, 75.136]
  MoveC 3919 to (-76.1, 59.76, -6) mm, rotated rx -180 ry 0 rz 90 deg; joints [75.1, -19.081, 90.833, 0, 18.247, 75.1] to (-76.17, 58.75, -6) mm, rotated rx -180 ry 0 rz 90 deg; joints [75.065, -19.078, 90.82, 0, 18.258, 75.065]
  MoveL 3920 to (-76.17, 29.55, -6) mm, rotated rx -180 ry 0 rz 90 deg; joints [74.068, -18.962, 90.283, 0, 18.679, 74.068]
  MoveL 3921 to (-68.62, 29.55, -6) mm, rotated rx -180 ry 0 rz 90 deg; joints [74.141, -18.85, 89.778, 0, 19.073, 74.141]
  MoveL 3922 to (-68.62, 29.55, -3) mm, rotated rx -180 ry 0 rz 90 deg; joints [74.141, -19.007, 89.879, 0, 19.128, 74.141]
  Establecer velocidad (1000.0 mm/s)
  MoveL 3923 to (-68.62, 29.55, 10) mm, rotated rx 180 ry 0 rz 90 deg; joints [74.141, -19.688, 90.312, 0, 19.375, 74.141]
  Establecer velocidad (66.7 mm/s)
  MoveL 3924 to (-39.6, -29.27, 10) mm, rotated rx 180 ry 0 rz 90 deg; joints [72.474, -18.933, 87.143, 0, 21.791, 72.474]
  MoveL 3925 to (-39.6, -29.27, -2.75) mm, rotated rx 180 ry 0 rz 90 deg; joints [72.474, -18.276, 86.718, 0, 21.558, 72.474]
  MoveL 3926 to (-39.73, -27.76, -3.16) mm, rotated rx -180 ry 0 rz 90 deg; joints [72.522, -18.265, 86.746, 0, 21.519, 72.522]
  MoveL 3927 to (-40.22, -26.32, -3.56) mm, rotated rx -180 ry 0 rz 90 deg; joints [72.564, -18.26, 86.797, 0, 21.463, 72.564]
  MoveL 3928 to (-41.02, -25.03, -3.97) mm, rotated rx -180 ry 0 rz 90 deg; joints [72.598, -18.259, 86.866, 0, 21.393, 72.598]
  MoveL 3929 to (-42.09, -23.95, -4.37) mm, rotated rx 180 ry 0 rz 90 deg; joints [72.623, -18.262, 86.949, 0, 21.313, 72.623]
  MoveL 3930 to (-43.37, -23.12, -4.78) mm, rotated rx -180 ry 0 rz 90 deg; joints [72.636, -18.267, 87.041, 0, 21.226, 72.636]
  MoveL 3931 to (-44.8, -22.61, -5.19) mm, rotated rx 180 ry 0 rz 90 deg; joints [72.639, -18.272, 87.136, 0, 21.136, 72.639]
  MoveL 3932 to (-46.3, -22.42, -5.59) mm, rotated rx 180 ry 0 rz 90 deg; joints [72.63, -18.277, 87.229, 0, 21.048, 72.63]
  MoveL 3933 to (-47.81, -22.6, -6) mm, rotated rx 180 ry 0 rz 90 deg; joints [72.608, -18.28, 87.315, 0, 20.965, 72.608]
  MoveL 3934 to (-72.52, -27.85, -6) mm, rotated rx 180 ry 0 rz 90 deg; joints [72.175, -18.646, 88.873, 0, 19.773, 72.175]
  MoveC 3935 to (-75.15, -29.46, -6) mm, rotated rx 180 ry 0 rz 90 deg; joints [72.093, -18.678, 89.015, 0, 19.664, 72.093] to (-76.17, -32.37, -6) mm, rotated rx 180 ry 0 rz 90 deg; joints [71.986, -18.68, 89.02, 0, 19.659, 71.986]
  MoveL 3936 to (-76.17, -71.01, -6) mm, rotated rx 180 ry 0 rz 90 deg; joints [70.71, -18.478, 88.148, 0, 20.33, 70.71]
  MoveC 3937 to (-75.78, -72.86, -6) mm, rotated rx 180 ry 0 rz 90 deg; joints [70.654, -18.461, 88.078, 0, 20.383, 70.654] to (-74.67, -74.39, -6) mm, rotated rx -180 ry 0 rz 90 deg; joints [70.617, -18.435, 87.968, 0, 20.468, 70.617]
  MoveC 3938 to (-73.03, -75.27, -6) mm, rotated rx 180 ry 0 rz 90 deg; joints [70.607, -18.404, 87.837, 0, 20.567, 70.607] to (-71.2, -75.55, -6) mm, rotated rx 180 ry 0 rz 90 deg; joints [70.619, -18.374, 87.707, 0, 20.667, 70.619]
  MoveL 3939 to (-35.33, -75.26, -6) mm, rotated rx -180 ry 0 rz 90 deg; joints [71.032, -17.773, 85.268, 0, 22.505, 71.032]
  MoveC 3940 to (-32.46, -74.26, -6) mm, rotated rx 180 ry 0 rz 90 deg; joints [71.095, -17.728, 85.093, 0, 22.635, 71.095] to (-30.79, -71.72, -6) mm, rotated rx 180 ry 0 rz 90 deg; joints [71.195, -17.714, 85.037, 0, 22.677, 71.195]
  MoveL 3941 to (-18.15, -23.22, -6) mm, rotated rx -180 ry 0 rz 90 deg; joints [72.888, -17.769, 85.252, 0, 22.517, 72.888]
  MoveC 3942 to (-17.98, -22.27, -6) mm, rotated rx -180 ry 0 rz 90 deg; joints [72.921, -17.771, 85.261, 0, 22.511, 72.921] to (-17.96, -21.3, -6) mm, rotated rx 180 ry 0 rz 90 deg; joints [72.952, -17.776, 85.28, 0, 22.496, 72.952]
  MoveC 3943 to (-19.61, -18.13, -6) mm, rotated rx 180 ry 0 rz 90 deg; joints [73.039, -17.823, 85.463, 0, 22.359, 73.039] to (-23.1, -17.34, -6) mm, rotated rx -180 ry 0 rz 90 deg; joints [73.03, -17.888, 85.723, 0, 22.165, 73.03]
  MoveL 3944 to (-47.81, -22.6, -6) mm, rotated rx 180 ry 0 rz 90 deg; joints [72.608, -18.28, 87.315, 0, 20.965, 72.608]
